// TwinCAT 3 PLC project MS
// ProgramVersion: 3.1.4024.0
// libraries:
//   Tc2_ControllerToolbox, * (Beckhoff Automation GmbH)
//   Tc2_ModbusRTU, * (Beckhoff Automation GmbH)
//   Tc2_SerialCom, * (Beckhoff Automation GmbH)
//   Tc2_Standard, * (Beckhoff Automation GmbH)
//   Tc2_System, * (Beckhoff Automation GmbH)
//   Tc2_Utilities, * (Beckhoff Automation GmbH)
//   Tc3_Module, * (Beckhoff Automation GmbH)
// project tree:
//   DATA TYPES/MODUELS/ ST_GAS_CABINET.TcDUT (not stored), ST_MAIN_MODULE.TcDUT (not stored), ST_NOTIFICATION.TcDUT (not stored), ST_NOTIFICATION_MESSAGE.TcDUT (not stored), ST_REACTOR_CABINET.TcDUT (not stored), ST_SEQUENCE.TcDUT (not stored), ST_SOL_VALVE.TcDUT (not stored), ST_TEMP_CONTROLLER.TcDUT (not stored), ST_THROTTLE_VALVE.TcDUT (not stored)
//   DATA TYPES/PARTS/ ST_ANALOG_PART.TcDUT (not stored), ST_DIGITAL_PART.TcDUT (not stored), ST_SEQUENCE_PART.TcDUT (not stored)
//   DEVICE/LINE HEATER/ FB_LINE_HEATER_MANAGER.TcPOU (not stored), FB_Modbus_Send_FIFO.TcPOU (not stored), FB_TEMP_RAMPING.TcPOU (not stored)
//   DEVICE/LINE HEATER/FUNCTION/ F_Temp_Write_Set_Point.TcPOU (not stored), F_Temp_Write_Value.TcPOU (not stored)
//   DEVICE/ ST_LineHeater_Data.TcDUT (not stored), ST_Modbus_Send_Frame.TcDUT (not stored)
//   DUTs/DUTs/ENUM/ E_aAnalogInputIO_Index.TcDUT, E_AlarmList.TcDUT (not stored), E_AlarmSetValue.TcDUT, E_InputState.TcDUT (not stored), E_Interlock.TcDUT (not stored), E_Morning_Index.TcDUT, E_WarningList.TcDUT (not stored)
//   DUTs/DUTs/ F_GetReal_USINT.TcDUT (not stored)
//   DUTs/ E_ControlMode.TcDUT (not stored), E_RampGeneratorState.TcDUT (not stored), E_RecipeRun.TcDUT (not stored), E_RecipeRunETMode.TcDUT (not stored), E_TowerLamp.TcDUT (not stored), OperationMode.TcDUT (not stored), outWord.TcDUT (not stored), RampGeneratorInput.TcDUT (not stored), RecipeRunET.TcDUT (not stored), RecipeStep.TcDUT, ScaleFactor.TcDUT (not stored)
//   FUNCTION/ BOOL_TO_STRING_LHeaterON.TcPOU (not stored), CheckRangeSigned.TcPOU (not stored), CheckRangeUnsigned.TcPOU (not stored), FB_TON_Pausable.TcPOU (not stored), F_GetDorPressure.TcPOU, F_State_All_Valve_Vent.TcPOU (not stored), HEXSTR_TO_REAL_LHeaterPV.TcPOU (not stored), Real_To_String_LineHeater.TcPOU (not stored), Real_To_String_ThermalBath.TcPOU (not stored), USINT_TO_WORD_Bit.TcPOU (not stored), USINT_TO_WORD_jh.TcPOU (not stored), WORD_TO_USINT_Bit.TcPOU (not stored)
//   GVLs/ GVL_COMMAND_FROM_UI.TcGVL (not stored), GVL_CONSTANT.TcGVL, GVL_DEVICE_NET_E3508.TcGVL, GVL_DEVICE_NET_IQ_PLUS.TcGVL (not stored), GVL_IO.TcGVL, GVL.TcGVL, GVL_IO_GAS_CABINET.TcGVL (not stored), GVL_IO_REACTOR_CABINET.TcGVL (not stored), GVL_IO_VALVE.TcGVL (not stored), GVL_PERSISTENT.TcGVL (not stored), GVL_SEQUENCE.TcGVL, GVL_Serial.TcGVL, RCP.TcGVL (not stored)
//   / PlcTask.TcTTO (not stored)
//   POUs/ FB_AnalogDeviceRampControl.TcPOU, FB_ControlRampGenerator.TcPOU (not stored), FB_DeviationCheck.TcPOU, FB_FaultCheck.TcPOU (not stored), FB_OnlyPVUpdate.TcPOU, FB_OverLimitCheck.TcPOU (not stored), FB_RecipeAnalogControlInputSequencer.TcPOU, F_StopAnalogRamping_ForRecipe.TcPOU, FB_SensorLimitCheck.TcPOU (not stored), FB_ValveControl.TcPOU, F_ResetTimersAndRCPTimes.TcPOU (not stored), MAIN.TcPOU, P11_E3508.TcPOU, P12_IQ_PLUS.TcPOU, P13_LineHeater.TcPOU, P14_ThermalBath.TcPOU, P15_RotationOperation.TcPOU, P16_CoverOperation.TcPOU, P17_DOROperation.TcPOU, P22_Background_ThermalBath.TcPOU (not stored), P30_ManualControl.TcPOU, P31_PriorityControl.TcPOU (not stored), P50_RecipeControl.TcPOU, P70_Interface.TcPOU, P90_Interlock.TcPOU, P91_Monitoring.TcPOU, P92_Maintenance.TcPOU
//   POUs/FUNCTION/ FB_RINGBUFFER.TcPOU (not stored), F_StateValve_Process_Source.TcPOU (not stored), F_StateValve_Process.TcPOU (not stored)
//   POUs/VARIABLE_LINK/ F_Variable_DeviceLink.TcPOU, F_Variable_Valve.TcPOU, F_Variable_FromUI.TcPOU, F_Variable_FromUI_Interlock.TcPOU, F_Variable_TODevice.TcPOU (not stored), F_Variable_ToUI_InputState.TcPOU
// real-time tasks:
//   TASK PlcTask: cycle T#10ms, priority 20, ADS port 350
// I/O:
//   DEVICE Device 1 (EtherCAT), AmsNetId 10.10.10.10.2.1
//     Term 1 (EK1200) [EK1200-5000 EtherCAT Power supply (2A E-Bus)]
//       Term 2 (EL1088) [EL1088 8Ch. Dig. Input 24V, 3ms, negative]
//       Term 3 (EL1088) [EL1088 8Ch. Dig. Input 24V, 3ms, negative]
//       Term 4 (EL1088) [EL1088 8Ch. Dig. Input 24V, 3ms, negative]
//       Term 5 (EL1088) [EL1088 8Ch. Dig. Input 24V, 3ms, negative]
//       Term 6 (EL1088) [EL1088 8Ch. Dig. Input 24V, 3ms, negative]
//       Term 7 (EL1088) [EL1088 8Ch. Dig. Input 24V, 3ms, negative]
//       Term 8 (EL2088) [EL2088 8Ch. Dig. Output 24V, 0.5A, switching to negative]
//       Term 9 (EL2088) [EL2088 8Ch. Dig. Output 24V, 0.5A, switching to negative]
//       Term 10 (EL3064) [EL3064 4Ch. Ana. Input 0-10V]
//       Term 11 (EL4004) [EL4004 4Ch. Ana. Output 0-10V, 12bit]
//       Term 12 (EL9410) [EL9410 E-Bus Power Supplier  (Diagnostics)]
//       Term 13 (EL3064) [EL3064 4Ch. Ana. Input 0-10V]
//       Term 14 (EL4004) [EL4004 4Ch. Ana. Output 0-10V, 12bit]
//       Term 15 (EL3064) [EL3064 4Ch. Ana. Input 0-10V]
//       Term 16 (EL4004) [EL4004 4Ch. Ana. Output 0-10V, 12bit]
//       Term 17 (EL3064) [EL3064 4Ch. Ana. Input 0-10V]
//       Term 18 (EL4004) [EL4004 4Ch. Ana. Output 0-10V, 12bit]
//       Term 19 (EL3102) [EL3102 2Ch. Ana. Input +/-10V, Diff.]
//       Term 20 (EL3024) [EL3024 4Ch. Ana. Input 4-20mA DIFF]
//       Term 21 (EL6021) [EL6021 Interface (RS422/485)]
//       Term 22 (EL6021) [EL6021 Interface (RS422/485)]
//       Term 23 (EL6752) [EL6752 DeviceNet Master]
//       Term 24 (EK1110) [EK1110 EtherCAT extension]
//     Term 25 (EK1100) [EK1100 EtherCAT Coupler (2A E-Bus)]
//       Term 26 (EL1088) [EL1088 8Ch. Dig. Input 24V, 3ms, negative]
//       Term 27 (EL1088) [EL1088 8Ch. Dig. Input 24V, 3ms, negative]
//       Term 28 (EL1088) [EL1088 8Ch. Dig. Input 24V, 3ms, negative]
//       Term 29 (EL2088) [EL2088 8Ch. Dig. Output 24V, 0.5A, switching to negative]
//       Term 30 (EL2088) [EL2088 8Ch. Dig. Output 24V, 0.5A, switching to negative]
//       Term 31 (EL2088) [EL2088 8Ch. Dig. Output 24V, 0.5A, switching to negative]
//       Term 32 (EL3064) [EL3064 4Ch. Ana. Input 0-10V]
//       Term 33 (EL3024) [EL3024 4Ch. Ana. Input 4-20mA DIFF]
//       Term 34 (EL4004) [EL4004 4Ch. Ana. Output 0-10V, 12bit]
//       Term 35 (EL3204) [EL3204 4Ch. Ana. Input PT100 (RTD)]
//       Term 36 (EL9011) [EL9011 End Terminal]
//   DEVICE Device 2 (EL6752), AmsNetId 10.10.10.10.3.1
//     SolValve // EDS-File: 'OPP6-2D.EDS' DescText: OPP6-2D Vendor: CKD Corporation Device Type: Generic Device Product Name: OPP6-2D Catalog Number:
//     ThrottleValve // EDS-File: 'TBJQPDNG-L041X01 155OUT154.EDS' DescText: Intellisys IQ-Plus Vendor: Nor-Cal Products Device Type: Process Control Valve Product Name: INTELLISYS Catalog Number: IQ-Plus
//     TempController // EDS-File: '3500-2.3V2.EDS' DescText: Eurotherm 3500 Vendor: Eurotherm Device Type: Generic Product Name: Eurotherm 3500 Catalog Number:
// variable links:
//   MS/MS Instance <-> Device 1 (EtherCAT)/Term 1 (EK1200)/Term 10 (EL3064)
//     PlcTask Inputs/GVL_IO_GAS_CABINET.AI_09_M01_ChalcogenRunPV <-> AI Standard Channel 1/Value
//     PlcTask Inputs/GVL_IO_GAS_CABINET.AI_09_M02_MORunPV <-> AI Standard Channel 2/Value
//     PlcTask Inputs/GVL_IO_GAS_CABINET.AI_09_M03_H2SeSupplyPV <-> AI Standard Channel 3/Value
//     PlcTask Inputs/GVL_IO_GAS_CABINET.AI_09_M04_H2SSupplyPV <-> AI Standard Channel 4/Value
//   MS/MS Instance <-> Device 1 (EtherCAT)/Term 1 (EK1200)/Term 11 (EL4004)
//     PlcTask Outputs/GVL_IO_GAS_CABINET.AO_10_M01_ChalcogenRunSV <-> AO Outputs Channel 1/Analog output
//     PlcTask Outputs/GVL_IO_GAS_CABINET.AO_10_M02_MORunSV <-> AO Outputs Channel 2/Analog output
//     PlcTask Outputs/GVL_IO_GAS_CABINET.AO_10_M03_H2SeSupplySV <-> AO Outputs Channel 3/Analog output
//     PlcTask Outputs/GVL_IO_GAS_CABINET.AO_10_M04_H2SSupplySV <-> AO Outputs Channel 4/Analog output
//   MS/MS Instance <-> Device 1 (EtherCAT)/Term 1 (EK1200)/Term 13 (EL3064)
//     PlcTask Inputs/GVL_IO_GAS_CABINET.AI_11_M05_Source_1TMInSupplyPV <-> AI Standard Channel 1/Value
//     PlcTask Inputs/GVL_IO_GAS_CABINET.AI_11_M06_Source_2TMGaSupplyPV <-> AI Standard Channel 2/Value
//     PlcTask Inputs/GVL_IO_GAS_CABINET.AI_11_M07_Source_3DMSeSupplyPV <-> AI Standard Channel 3/Value
//     PlcTask Inputs/GVL_IO_GAS_CABINET.AI_11_M08_Source_4ChalcoSupplyPV <-> AI Standard Channel 4/Value
//   MS/MS Instance <-> Device 1 (EtherCAT)/Term 1 (EK1200)/Term 14 (EL4004)
//     PlcTask Outputs/GVL_IO_GAS_CABINET.AO_12_M05_Source_1TMInSupplySV <-> AO Outputs Channel 1/Analog output
//     PlcTask Outputs/GVL_IO_GAS_CABINET.AO_12_M06_Source_2TMGaSupplySV <-> AO Outputs Channel 2/Analog output
//     PlcTask Outputs/GVL_IO_GAS_CABINET.AO_12_M07_Source_3DMSeSupplySV <-> AO Outputs Channel 3/Analog output
//     PlcTask Outputs/GVL_IO_GAS_CABINET.AO_12_M08_Source_4ChalcoSupplySV <-> AO Outputs Channel 4/Analog output
//   MS/MS Instance <-> Device 1 (EtherCAT)/Term 1 (EK1200)/Term 15 (EL3064)
//     PlcTask Inputs/GVL_IO_GAS_CABINET.AI_13_M09_LinerPurgePV <-> AI Standard Channel 1/Value
//     PlcTask Inputs/GVL_IO_GAS_CABINET.AI_13_M10_HeaterPurgePV <-> AI Standard Channel 2/Value
//     PlcTask Inputs/GVL_IO_GAS_CABINET.AI_13_M11_ChalcogenVentPV <-> AI Standard Channel 3/Value
//     PlcTask Inputs/GVL_IO_GAS_CABINET.AI_13_M12_MOVentPV <-> AI Standard Channel 4/Value
//   MS/MS Instance <-> Device 1 (EtherCAT)/Term 1 (EK1200)/Term 16 (EL4004)
//     PlcTask Outputs/GVL_IO_GAS_CABINET.AO_14_M09_LinerPurgeSV <-> AO Outputs Channel 1/Analog output
//     PlcTask Outputs/GVL_IO_GAS_CABINET.AO_14_M10_HeaterPurgeSV <-> AO Outputs Channel 2/Analog output
//     PlcTask Outputs/GVL_IO_GAS_CABINET.AO_14_M11_ChalcogenVentSV <-> AO Outputs Channel 3/Analog output
//     PlcTask Outputs/GVL_IO_GAS_CABINET.AO_14_M12_MOVentSV <-> AO Outputs Channel 4/Analog output
//   MS/MS Instance <-> Device 1 (EtherCAT)/Term 1 (EK1200)/Term 17 (EL3064)
//     PlcTask Inputs/GVL_IO_GAS_CABINET.AI_15_E01Source_1TMInPressurePV <-> AI Standard Channel 1/Value
//     PlcTask Inputs/GVL_IO_GAS_CABINET.AI_15_E02Source_2TMGaPressurePV <-> AI Standard Channel 2/Value
//     PlcTask Inputs/GVL_IO_GAS_CABINET.AI_15_E03Source_3DMSePressurePV <-> AI Standard Channel 3/Value
//     PlcTask Inputs/GVL_IO_GAS_CABINET.AI_15_E04Source_4ChalcoPressurePV <-> AI Standard Channel 4/Value
//   MS/MS Instance <-> Device 1 (EtherCAT)/Term 1 (EK1200)/Term 18 (EL4004)
//     PlcTask Outputs/GVL_IO_GAS_CABINET.AO_16_E01Source_1TMInPressureSV <-> AO Outputs Channel 1/Analog output
//     PlcTask Outputs/GVL_IO_GAS_CABINET.AO_16_E02Source_2TMGaPressureSV <-> AO Outputs Channel 2/Analog output
//     PlcTask Outputs/GVL_IO_GAS_CABINET.AO_16_E03Source_3DMSePressureSV <-> AO Outputs Channel 3/Analog output
//     PlcTask Outputs/GVL_IO_GAS_CABINET.AO_16_E04Source_4ChalcoPressureSV <-> AO Outputs Channel 4/Analog output
//   MS/MS Instance <-> Device 1 (EtherCAT)/Term 1 (EK1200)/Term 19 (EL3102)
//     PlcTask Inputs/GVL_IO_GAS_CABINET.DI_17_DP1ChalcogenDP <-> AI Standard Channel 1/Value
//     PlcTask Inputs/GVL_IO_GAS_CABINET.DI_17_DP2MODP <-> AI Standard Channel 2/Value
//   MS/MS Instance <-> Device 1 (EtherCAT)/Term 1 (EK1200)/Term 2 (EL1088)
//     PlcTask Inputs/GVL_IO_GAS_CABINET.DI_01_ControlCabinetDoorClose <-> Channel 5/Input
//     PlcTask Inputs/GVL_IO_GAS_CABINET.DI_01_GasCabinetDoorClose <-> Channel 4/Input
//     PlcTask Inputs/GVL_IO_GAS_CABINET.DI_01_GasCabinetLampButton <-> Channel 2/Input
//     PlcTask Inputs/GVL_IO_GAS_CABINET.DI_01_PneumaticPressureSensor <-> Channel 3/Input
//     PlcTask Inputs/GVL_IO_GAS_CABINET.DI_01_ResetButton <-> Channel 1/Input
//     PlcTask Inputs/GVL_IO_GAS_CABINET.DI_01_SMPS_1Alarm <-> Channel 6/Input
//     PlcTask Inputs/GVL_IO_GAS_CABINET.DI_01_SMPS_2Alarm <-> Channel 7/Input
//     PlcTask Inputs/GVL_IO_GAS_CABINET.DI_01_SMPS_3Alarm <-> Channel 8/Input
//   MS/MS Instance <-> Device 1 (EtherCAT)/Term 1 (EK1200)/Term 20 (EL3024)
//     PlcTask Inputs/GVL_IO_GAS_CABINET.DI_18_S01N2SupplyPressPV <-> AI Standard Channel 1/Value
//     PlcTask Inputs/GVL_IO_GAS_CABINET.DI_18_S02H2SupplyPressPV <-> AI Standard Channel 2/Value
//     PlcTask Inputs/GVL_IO_GAS_CABINET.DI_18_S03H2SSupplyPressPV <-> AI Standard Channel 3/Value
//     PlcTask Inputs/GVL_IO_GAS_CABINET.DI_18_S04H2SeSupplyPressPV <-> AI Standard Channel 4/Value
//   MS/MS Instance <-> Device 1 (EtherCAT)/Term 1 (EK1200)/Term 21 (EL6021)
//     PlcTask Inputs/GVL.fbLineHeater_Manager.fbModbus_Master.InData/D <-> COM TxPDO-Map Inputs/Data In 0
//     PlcTask Inputs/GVL.fbLineHeater_Manager.fbModbus_Master.InData/D @bit {8..168 step 8} <-> COM TxPDO-Map Inputs/Data In {1..21}  (21 links)
//     PlcTask Inputs/GVL.fbLineHeater_Manager.fbModbus_Master.InData/Status <-> COM TxPDO-Map Inputs/Status
//     PlcTask Outputs/GVL.fbLineHeater_Manager.fbModbus_Master.OutData/Ctrl <-> COM RxPDO-Map Outputs/Ctrl
//     PlcTask Outputs/GVL.fbLineHeater_Manager.fbModbus_Master.OutData/D <-> COM RxPDO-Map Outputs/Data Out 0
//     PlcTask Outputs/GVL.fbLineHeater_Manager.fbModbus_Master.OutData/D @bit {8..168 step 8} <-> COM RxPDO-Map Outputs/Data Out {1..21}  (21 links)
//   MS/MS Instance <-> Device 1 (EtherCAT)/Term 1 (EK1200)/Term 22 (EL6021)
//     PlcTask Inputs/GVL_Serial.stIn_KL6031_TB/D <-> COM TxPDO-Map Inputs/Data In 0
//     PlcTask Inputs/GVL_Serial.stIn_KL6031_TB/D @bit {8..168 step 8} <-> COM TxPDO-Map Inputs/Data In {1..21}  (21 links)
//     PlcTask Inputs/GVL_Serial.stIn_KL6031_TB/Status <-> COM TxPDO-Map Inputs/Status
//     PlcTask Outputs/GVL_Serial.stOut_KL6031_TB/Ctrl <-> COM RxPDO-Map Outputs/Ctrl
//     PlcTask Outputs/GVL_Serial.stOut_KL6031_TB/D <-> COM RxPDO-Map Outputs/Data Out 0
//     PlcTask Outputs/GVL_Serial.stOut_KL6031_TB/D @bit {8..168 step 8} <-> COM RxPDO-Map Outputs/Data Out {1..21}  (21 links)
//   MS/MS Instance <-> Device 1 (EtherCAT)/Term 1 (EK1200)/Term 3 (EL1088)
//     PlcTask Inputs/GVL_IO_GAS_CABINET.DI_02_CoverLiftMotorCP <-> Channel 7/Input
//     PlcTask Inputs/GVL_IO_GAS_CABINET.DI_02_GraphiteHeaterELCB <-> Channel 2/Input
//     PlcTask Inputs/GVL_IO_GAS_CABINET.DI_02_LineHeatersELCB <-> Channel 5/Input
//     PlcTask Inputs/GVL_IO_GAS_CABINET.DI_02_RotationMotorCP <-> Channel 6/Input
//     PlcTask Inputs/GVL_IO_GAS_CABINET.DI_02_SMPS_4Alarm <-> Channel 1/Input
//     PlcTask Inputs/GVL_IO_GAS_CABINET.DI_02_T_VCP <-> Channel 8/Input
//     PlcTask Inputs/GVL_IO_GAS_CABINET.DI_02_ThermalBathsELCB <-> Channel 3/Input
//     PlcTask Inputs/GVL_IO_GAS_CABINET.DI_02_VacuumPumpELCB <-> Channel 4/Input
//   MS/MS Instance <-> Device 1 (EtherCAT)/Term 1 (EK1200)/Term 4 (EL1088)
//     PlcTask Inputs/GVL_IO_GAS_CABINET.DI_03_CabinetLampsCP <-> Channel 2/Input
//     PlcTask Inputs/GVL_IO_GAS_CABINET.DI_03_GasDetectorCP <-> Channel 1/Input
//     PlcTask Inputs/GVL_IO_GAS_CABINET.DI_03_LineHeater_1CP <-> Channel 4/Input
//     PlcTask Inputs/GVL_IO_GAS_CABINET.DI_03_LineHeater_2CP <-> Channel 5/Input
//     PlcTask Inputs/GVL_IO_GAS_CABINET.DI_03_LineHeater_3CP <-> Channel 6/Input
//     PlcTask Inputs/GVL_IO_GAS_CABINET.DI_03_LineHeater_4CP <-> Channel 7/Input
//     PlcTask Inputs/GVL_IO_GAS_CABINET.DI_03_LineHeater_5CP <-> Channel 8/Input
//     PlcTask Inputs/GVL_IO_GAS_CABINET.DI_03_MFCPowerCP <-> Channel 3/Input
//   MS/MS Instance <-> Device 1 (EtherCAT)/Term 1 (EK1200)/Term 5 (EL1088)
//     PlcTask Inputs/GVL_IO_GAS_CABINET.DI_04_ExternalScrubberFault <-> Channel 8/Input
//     PlcTask Inputs/GVL_IO_GAS_CABINET.DI_04_FireSensor <-> Channel 7/Input
//     PlcTask Inputs/GVL_IO_GAS_CABINET.DI_04_GasDetectorH2 <-> Channel 4/Input
//     PlcTask Inputs/GVL_IO_GAS_CABINET.DI_04_GasDetectorH2S <-> Channel 5/Input
//     PlcTask Inputs/GVL_IO_GAS_CABINET.DI_04_GasDetectorH2Se <-> Channel 6/Input
//     PlcTask Inputs/GVL_IO_GAS_CABINET.DI_04_LineHeater_6CP <-> Channel 1/Input
//     PlcTask Inputs/GVL_IO_GAS_CABINET.DI_04_LineHeater_7CP <-> Channel 2/Input
//     PlcTask Inputs/GVL_IO_GAS_CABINET.DI_04_LineHeater_8CP <-> Channel 3/Input
//   MS/MS Instance <-> Device 1 (EtherCAT)/Term 1 (EK1200)/Term 6 (EL1088)
//     PlcTask Inputs/GVL_IO_GAS_CABINET.DI_05_ExternalH2GasCabinetFault <-> Channel 1/Input
//     PlcTask Inputs/GVL_IO_GAS_CABINET.DI_05_ExternalH2SGasCabinetFault <-> Channel 2/Input
//     PlcTask Inputs/GVL_IO_GAS_CABINET.DI_05_ExternalH2SeGasCabinetFault <-> Channel 3/Input
//     PlcTask Inputs/GVL_IO_GAS_CABINET.DI_05_ExternalUserInputAlarm <-> Channel 4/Input
//     PlcTask Inputs/GVL_IO_GAS_CABINET.DI_05_ThermalBath_1CutOffAlarm <-> Channel 6/Input
//     PlcTask Inputs/GVL_IO_GAS_CABINET.DI_05_ThermalBath_2CutOffAlarm <-> Channel 8/Input
//     PlcTask Inputs/GVL_IO_GAS_CABINET.DI_05_ThermalBath_1DeviationAlarm <-> Channel 5/Input
//     PlcTask Inputs/GVL_IO_GAS_CABINET.DI_05_ThermalBath_2DeviationAlarm <-> Channel 7/Input
//   MS/MS Instance <-> Device 1 (EtherCAT)/Term 1 (EK1200)/Term 7 (EL1088)
//     PlcTask Inputs/GVL_IO_GAS_CABINET.DI_06_Spare_01 <-> Channel 5/Input
//     PlcTask Inputs/GVL_IO_GAS_CABINET.DI_06_Spare_02 <-> Channel 6/Input
//     PlcTask Inputs/GVL_IO_GAS_CABINET.DI_06_Spare_03 <-> Channel 7/Input
//     PlcTask Inputs/GVL_IO_GAS_CABINET.DI_06_Spare_04 <-> Channel 8/Input
//     PlcTask Inputs/GVL_IO_GAS_CABINET.DI_06_ThermalBath_3CutOffAlarm <-> Channel 2/Input
//     PlcTask Inputs/GVL_IO_GAS_CABINET.DI_06_ThermalBath_4CutOffAlarm <-> Channel 4/Input
//     PlcTask Inputs/GVL_IO_GAS_CABINET.DI_06_ThermalBath_3DeviationAlarm <-> Channel 1/Input
//     PlcTask Inputs/GVL_IO_GAS_CABINET.DI_06_ThermalBath_4DeviationAlarm <-> Channel 3/Input
//   MS/MS Instance <-> Device 1 (EtherCAT)/Term 1 (EK1200)/Term 8 (EL2088)
//     PlcTask Outputs/GVL_IO_GAS_CABINET.DO_07_ControlCabinetLamp <-> Channel 2/Output
//     PlcTask Outputs/GVL_IO_GAS_CABINET.DO_07_GasCabinetLamp <-> Channel 3/Output
//     PlcTask Outputs/GVL_IO_GAS_CABINET.DO_07_GraphiteHeaterMC <-> Channel 4/Output
//     PlcTask Outputs/GVL_IO_GAS_CABINET.DO_07_LineHeatersMC <-> Channel 7/Output
//     PlcTask Outputs/GVL_IO_GAS_CABINET.DO_07_ResetButtonLamp <-> Channel 8/Output
//     PlcTask Outputs/GVL_IO_GAS_CABINET.DO_07_SystemPowerOffLock <-> Channel 1/Output
//     PlcTask Outputs/GVL_IO_GAS_CABINET.DO_07_ThermalBathsMC <-> Channel 5/Output
//     PlcTask Outputs/GVL_IO_GAS_CABINET.DO_07_VacuumPumpMC <-> Channel 6/Output
//   MS/MS Instance <-> Device 1 (EtherCAT)/Term 1 (EK1200)/Term 9 (EL2088)
//     PlcTask Outputs/GVL_IO_GAS_CABINET.DO_08_Spare_01 <-> Channel 1/Output
//     PlcTask Outputs/GVL_IO_GAS_CABINET.DO_08_Spare_02 <-> Channel 2/Output
//     PlcTask Outputs/GVL_IO_GAS_CABINET.DO_08_Spare_03 <-> Channel 3/Output
//     PlcTask Outputs/GVL_IO_GAS_CABINET.DO_08_Spare_04 <-> Channel 4/Output
//     PlcTask Outputs/GVL_IO_GAS_CABINET.DO_08_Spare_05 <-> Channel 5/Output
//     PlcTask Outputs/GVL_IO_GAS_CABINET.DO_08_Spare_06 <-> Channel 6/Output
//     PlcTask Outputs/GVL_IO_GAS_CABINET.DO_08_Spare_07 <-> Channel 7/Output
//     PlcTask Outputs/GVL_IO_GAS_CABINET.DO_08_Spare_08 <-> Channel 8/Output
//   MS/MS Instance <-> Device 1 (EtherCAT)/Term 25 (EK1100)/Term 26 (EL1088)
//     PlcTask Inputs/GVL_IO_REACTOR_CABINET.DI_01_ClampLock <-> Channel 7/Input
//     PlcTask Inputs/GVL_IO_REACTOR_CABINET.DI_01_ClampRelease <-> Channel 8/Input
//     PlcTask Inputs/GVL_IO_REACTOR_CABINET.DI_01_DORATMButton <-> Channel 4/Input
//     PlcTask Inputs/GVL_IO_REACTOR_CABINET.DI_01_DORVACButton <-> Channel 3/Input
//     PlcTask Inputs/GVL_IO_REACTOR_CABINET.DI_01_MaintenanceModeKey <-> Channel 1/Input
//     PlcTask Inputs/GVL_IO_REACTOR_CABINET.DI_01_ReactorCabinetLampButton <-> Channel 2/Input
//     PlcTask Inputs/GVL_IO_REACTOR_CABINET.DI_01_ReactorDoorDownButton <-> Channel 6/Input
//     PlcTask Inputs/GVL_IO_REACTOR_CABINET.DI_01_ReactorDoorUpButton <-> Channel 5/Input
//   MS/MS Instance <-> Device 1 (EtherCAT)/Term 25 (EK1100)/Term 27 (EL1088)
//     PlcTask Inputs/GVL_IO_REACTOR_CABINET.DI_02_C_WFlowSensor <-> Channel 1/Input
//     PlcTask Inputs/GVL_IO_REACTOR_CABINET.DI_02_ReactorDoorUpLimitSensor <-> Channel 8/Input
//     PlcTask Inputs/GVL_IO_REACTOR_CABINET.DI_02_SusceptorRotationMotorFault <-> Channel 2/Input
//     PlcTask Inputs/GVL_IO_REACTOR_CABINET.DI_02_VacuumPumpAlarm <-> Channel 5/Input
//     PlcTask Inputs/GVL_IO_REACTOR_CABINET.DI_02_VacuumPumpFBRunning <-> Channel 7/Input
//     PlcTask Inputs/GVL_IO_REACTOR_CABINET.DI_02_VacuumPumpFail <-> Channel 3/Input
//     PlcTask Inputs/GVL_IO_REACTOR_CABINET.DI_02_VacuumPumpRunning <-> Channel 6/Input
//     PlcTask Inputs/GVL_IO_REACTOR_CABINET.DI_02_VacuumPumpWarning <-> Channel 4/Input
//   MS/MS Instance <-> Device 1 (EtherCAT)/Term 25 (EK1100)/Term 28 (EL1088)
//     PlcTask Inputs/GVL_IO_REACTOR_CABINET.DI_03_CylinderAutoSwitch_Closed <-> Channel 2/Input
//     PlcTask Inputs/GVL_IO_REACTOR_CABINET.DI_03_CylinderAutoSwitch_Opened <-> Channel 3/Input
//     PlcTask Inputs/GVL_IO_REACTOR_CABINET.DI_03_ReactorCabinetDoorClose <-> Channel 4/Input
//     PlcTask Inputs/GVL_IO_REACTOR_CABINET.DI_03_ReactorDoorDownLimitSensor <-> Channel 1/Input
//     PlcTask Inputs/GVL_IO_REACTOR_CABINET.DI_03_Spare_01 <-> Channel 5/Input
//     PlcTask Inputs/GVL_IO_REACTOR_CABINET.DI_03_Spare_02 <-> Channel 6/Input
//     PlcTask Inputs/GVL_IO_REACTOR_CABINET.DI_03_Spare_03 <-> Channel 7/Input
//     PlcTask Inputs/GVL_IO_REACTOR_CABINET.DI_03_Spare_04 <-> Channel 8/Input
//   MS/MS Instance <-> Device 1 (EtherCAT)/Term 25 (EK1100)/Term 29 (EL2088)
//     PlcTask Outputs/GVL_IO_REACTOR_CABINET.DO_04_ReactorCoverDownRelay <-> Channel 8/Output
//     PlcTask Outputs/GVL_IO_REACTOR_CABINET.DO_04_ReactorCoverUpRelay <-> Channel 7/Output
//     PlcTask Outputs/GVL_IO_REACTOR_CABINET.DO_04_SignalTowerBlue <-> Channel 4/Output
//     PlcTask Outputs/GVL_IO_REACTOR_CABINET.DO_04_SignalTowerBuzzer <-> Channel 6/Output
//     PlcTask Outputs/GVL_IO_REACTOR_CABINET.DO_04_SignalTowerGreen <-> Channel 3/Output
//     PlcTask Outputs/GVL_IO_REACTOR_CABINET.DO_04_SignalTowerOrange <-> Channel 2/Output
//     PlcTask Outputs/GVL_IO_REACTOR_CABINET.DO_04_SignalTowerRed <-> Channel 1/Output
//     PlcTask Outputs/GVL_IO_REACTOR_CABINET.DO_04_SignalTowerWhite <-> Channel 5/Output
//   MS/MS Instance <-> Device 1 (EtherCAT)/Term 25 (EK1100)/Term 30 (EL2088)
//     PlcTask Outputs/GVL_IO_REACTOR_CABINET.DO_05_ClampLock <-> Channel 1/Output
//     PlcTask Outputs/GVL_IO_REACTOR_CABINET.DO_05_ClampRelease <-> Channel 2/Output
//     PlcTask Outputs/GVL_IO_REACTOR_CABINET.DO_05_DORVACButtonLamp <-> Channel 8/Output
//     PlcTask Outputs/GVL_IO_REACTOR_CABINET.DO_05_SusceptorRotationAL_RST <-> Channel 7/Output
//     PlcTask Outputs/GVL_IO_REACTOR_CABINET.DO_05_SusceptorRotationFWD <-> Channel 5/Output
//     PlcTask Outputs/GVL_IO_REACTOR_CABINET.DO_05_SusceptorRotationSTOP <-> Channel 6/Output
//     PlcTask Outputs/GVL_IO_REACTOR_CABINET.DO_05_VacuumPumpReset <-> Channel 4/Output
//     PlcTask Outputs/GVL_IO_REACTOR_CABINET.DO_05_VacuumPumpStart_Stop <-> Channel 3/Output
//   MS/MS Instance <-> Device 1 (EtherCAT)/Term 25 (EK1100)/Term 31 (EL2088)
//     PlcTask Outputs/GVL_IO_REACTOR_CABINET.DO_06_ClampLockButtonLamp <-> Channel 4/Output
//     PlcTask Outputs/GVL_IO_REACTOR_CABINET.DO_06_ClampReleaseButtonLamp <-> Channel 5/Output
//     PlcTask Outputs/GVL_IO_REACTOR_CABINET.DO_06_DORATMButtonLamp <-> Channel 1/Output
//     PlcTask Outputs/GVL_IO_REACTOR_CABINET.DO_06_ReactorCabinetLamp <-> Channel 6/Output
//     PlcTask Outputs/GVL_IO_REACTOR_CABINET.DO_06_ReactorCoverDownButtonLamp <-> Channel 3/Output
//     PlcTask Outputs/GVL_IO_REACTOR_CABINET.DO_06_ReactorCoverUpButtonLamp <-> Channel 2/Output
//     PlcTask Outputs/GVL_IO_REACTOR_CABINET.DO_06_Spare07 <-> Channel 7/Output
//     PlcTask Outputs/GVL_IO_REACTOR_CABINET.DO_06_Spare08 <-> Channel 8/Output
//   MS/MS Instance <-> Device 1 (EtherCAT)/Term 25 (EK1100)/Term 32 (EL3064)
//     PlcTask Inputs/GVL_IO_REACTOR_CABINET.AI_07_P02_ReactorPressure10TorrPV <-> AI Standard Channel 1/Value
//     PlcTask Inputs/GVL_IO_REACTOR_CABINET.AI_07_P03_ExhaustPressurePV <-> AI Standard Channel 3/Value
//     PlcTask Inputs/GVL_IO_REACTOR_CABINET.AI_07_S05_DORPressurePV <-> AI Standard Channel 2/Value
//     PlcTask Inputs/GVL_IO_REACTOR_CABINET.AI_07_Spare_04 <-> AI Standard Channel 4/Value
//   MS/MS Instance <-> Device 1 (EtherCAT)/Term 25 (EK1100)/Term 33 (EL3024)
//     PlcTask Inputs/GVL_IO_REACTOR_CABINET.AI_08_R01SusceptorRotationPV <-> AI Standard Channel 1/Value
//     PlcTask Inputs/GVL_IO_REACTOR_CABINET.AI_08_Spare_02 <-> AI Standard Channel 2/Value
//     PlcTask Inputs/GVL_IO_REACTOR_CABINET.AI_08_Spare_03 <-> AI Standard Channel 3/Value
//     PlcTask Inputs/GVL_IO_REACTOR_CABINET.AI_08_Spare_04 <-> AI Standard Channel 4/Value
//   MS/MS Instance <-> Device 1 (EtherCAT)/Term 25 (EK1100)/Term 34 (EL4004)
//     PlcTask Outputs/GVL_IO_REACTOR_CABINET.AO_09_P03_ExhaustPressureAM215Input <-> AO Outputs Channel 1/Analog output
//     PlcTask Outputs/GVL_IO_REACTOR_CABINET.AO_09_R01_SusceptorRotationSV <-> AO Outputs Channel 2/Analog output
//     PlcTask Outputs/GVL_IO_REACTOR_CABINET.AO_09_Spare_03 <-> AO Outputs Channel 3/Analog output
//     PlcTask Outputs/GVL_IO_REACTOR_CABINET.AO_09_Spare_04 <-> AO Outputs Channel 4/Analog output
//   MS/MS Instance <-> Device 1 (EtherCAT)/Term 25 (EK1100)/Term 35 (EL3204)
//     PlcTask Inputs/GVL_IO_REACTOR_CABINET.AI_10_R04S_HCoolingWaterPV <-> RTD Inputs Channel 1/Value
//     PlcTask Inputs/GVL_IO_REACTOR_CABINET.AI_10_Spare_02 <-> RTD Inputs Channel 2/Value
//     PlcTask Inputs/GVL_IO_REACTOR_CABINET.AI_10_Spare_03 <-> RTD Inputs Channel 3/Value
//     PlcTask Inputs/GVL_IO_REACTOR_CABINET.AI_10_Spare_04 <-> RTD Inputs Channel 4/Value
//   MS/MS Instance <-> Device 2 (EL6752)/SolValve
//     PlcTask Outputs/GVL_IO_VALVE.DO_00_V01ChalcogenCarrierChange <-> Connection (Poll)/Outputs/Output Data[0]
//     PlcTask Outputs/GVL_IO_VALVE.DO_00_V02MOCarreirChange <-> Connection (Poll)/Outputs/Output Data[0] @bit 1
//     PlcTask Outputs/GVL_IO_VALVE.DO_00_V03H2SeSourceChange <-> Connection (Poll)/Outputs/Output Data[0] @bit 2
//     PlcTask Outputs/GVL_IO_VALVE.DO_00_V04H2SSourceChange <-> Connection (Poll)/Outputs/Output Data[0] @bit 3
//     PlcTask Outputs/GVL_IO_VALVE.DO_00_V05Source_1TMInCarrierChange <-> Connection (Poll)/Outputs/Output Data[0] @bit 4
//     PlcTask Outputs/GVL_IO_VALVE.DO_00_V06Source_1TMInBypass <-> Connection (Poll)/Outputs/Output Data[0] @bit 5
//     PlcTask Outputs/GVL_IO_VALVE.DO_00_V07Source_2TMGaCarrierChange <-> Connection (Poll)/Outputs/Output Data[0] @bit 6
//     PlcTask Outputs/GVL_IO_VALVE.DO_00_V08Source_2TMGaBypass <-> Connection (Poll)/Outputs/Output Data[0] @bit 7
//     PlcTask Outputs/GVL_IO_VALVE.DO_00_V09Source_3DMSeCarrierChange <-> Connection (Poll)/Outputs/Output Data[1]
//     PlcTask Outputs/GVL_IO_VALVE.DO_00_V10Source_3DMSeBypass <-> Connection (Poll)/Outputs/Output Data[1] @bit 1
//     PlcTask Outputs/GVL_IO_VALVE.DO_00_V11Source_4ChalcogenCarrierChange <-> Connection (Poll)/Outputs/Output Data[1] @bit 2
//     PlcTask Outputs/GVL_IO_VALVE.DO_00_V12Source_4ChalcogenBypass <-> Connection (Poll)/Outputs/Output Data[1] @bit 3
//     PlcTask Outputs/GVL_IO_VALVE.DO_00_V13ReactorPurgeCarrierChange <-> Connection (Poll)/Outputs/Output Data[1] @bit 4
//     PlcTask Outputs/GVL_IO_VALVE.DO_00_V14Source_1TMInManifoldRun <-> Connection (Poll)/Outputs/Output Data[1] @bit 5
//     PlcTask Outputs/GVL_IO_VALVE.DO_00_V15Source_2TMGaManifoldRun <-> Connection (Poll)/Outputs/Output Data[1] @bit 6
//     PlcTask Outputs/GVL_IO_VALVE.DO_00_V16Source_3DMSeManifoldRun <-> Connection (Poll)/Outputs/Output Data[1] @bit 7
//     PlcTask Outputs/GVL_IO_VALVE.DO_00_V17GasH2SeManifoldRun <-> Connection (Poll)/Outputs/Output Data[2]
//     PlcTask Outputs/GVL_IO_VALVE.DO_00_V18GasH2SManifoldRun <-> Connection (Poll)/Outputs/Output Data[2] @bit 1
//     PlcTask Outputs/GVL_IO_VALVE.DO_00_V19Source_4ChalcogenManifoldRun <-> Connection (Poll)/Outputs/Output Data[2] @bit 2
//     PlcTask Outputs/GVL_IO_VALVE.DO_00_V20VentPress_Change <-> Connection (Poll)/Outputs/Output Data[2] @bit 3
//     PlcTask Outputs/GVL_IO_VALVE.DO_00_V21PumpByPass <-> Connection (Poll)/Outputs/Output Data[2] @bit 4
//     PlcTask Outputs/GVL_IO_VALVE.DO_00_V22DORVaccumON <-> Connection (Poll)/Outputs/Output Data[2] @bit 5
//     PlcTask Outputs/GVL_IO_VALVE.DO_00_V23DORFilling <-> Connection (Poll)/Outputs/Output Data[2] @bit 6
//     PlcTask Outputs/GVL_IO_VALVE.DO_00_V24Source_1LeakTest_IN <-> Connection (Poll)/Outputs/Output Data[2] @bit 7
//     PlcTask Outputs/GVL_IO_VALVE.DO_00_V26Source_2LeakTest_IN <-> Connection (Poll)/Outputs/Output Data[3] @bit 1
//     PlcTask Outputs/GVL_IO_VALVE.DO_00_V28Source_3LeakTest_IN <-> Connection (Poll)/Outputs/Output Data[3] @bit 3
//     PlcTask Outputs/GVL_IO_VALVE.DO_00_V30Source_4LeakTest_IN <-> Connection (Poll)/Outputs/Output Data[3] @bit 5
//     PlcTask Outputs/GVL_IO_VALVE.DO_00_V25Source_1LeakTest_OUT <-> Connection (Poll)/Outputs/Output Data[3]
//     PlcTask Outputs/GVL_IO_VALVE.DO_00_V27Source_2LeakTest_OUT <-> Connection (Poll)/Outputs/Output Data[3] @bit 2
//     PlcTask Outputs/GVL_IO_VALVE.DO_00_V29Source_3LeakTest_OUT <-> Connection (Poll)/Outputs/Output Data[3] @bit 4
//     PlcTask Outputs/GVL_IO_VALVE.DO_00_V31Source_4LeakTest_OUT <-> Connection (Poll)/Outputs/Output Data[3] @bit 6
//     PlcTask Outputs/GVL_IO_VALVE.DO_00_V32SourceVacuumON <-> Connection (Poll)/Outputs/Output Data[3] @bit 7
//   MS/MS Instance <-> Device 2 (EL6752)/TempController
//     PlcTask Inputs/GVL_DEVICE_NET_E3508.aInputActiveOut[1] <-> Connection (Poll)/Inputs/Input Data_5
//     PlcTask Inputs/GVL_DEVICE_NET_E3508.aInputActiveOut[2] <-> Connection (Poll)/Inputs/Input Data_6
//     PlcTask Inputs/GVL_DEVICE_NET_E3508.aInputAlarmStatus[1] <-> Connection (Poll)/Inputs/Input Data_7
//     PlcTask Inputs/GVL_DEVICE_NET_E3508.aInputAlarmStatus[2] <-> Connection (Poll)/Inputs/Input Data_8
//     PlcTask Inputs/GVL_DEVICE_NET_E3508.aInputDerivative[1] <-> Connection (Poll)/Inputs/Input Data_17
//     PlcTask Inputs/GVL_DEVICE_NET_E3508.aInputDerivative[2] <-> Connection (Poll)/Inputs/Input Data_18
//     PlcTask Inputs/GVL_DEVICE_NET_E3508.aInputIntegral[1] <-> Connection (Poll)/Inputs/Input Data_15
//     PlcTask Inputs/GVL_DEVICE_NET_E3508.aInputIntegral[2] <-> Connection (Poll)/Inputs/Input Data_16
//     PlcTask Inputs/GVL_DEVICE_NET_E3508.aInputManAutoBytes[1] <-> Connection (Poll)/Inputs/Input Data_9
//     PlcTask Inputs/GVL_DEVICE_NET_E3508.aInputManAutoBytes[2] <-> Connection (Poll)/Inputs/Input Data_10
//     PlcTask Inputs/GVL_DEVICE_NET_E3508.aInputPVBytes[1] <-> Connection (Poll)/Inputs/Input Data_1
//     PlcTask Inputs/GVL_DEVICE_NET_E3508.aInputPVBytes[2] <-> Connection (Poll)/Inputs/Input Data_2
//     PlcTask Inputs/GVL_DEVICE_NET_E3508.aInputProportional[1] <-> Connection (Poll)/Inputs/Input Data_13
//     PlcTask Inputs/GVL_DEVICE_NET_E3508.aInputProportional[2] <-> Connection (Poll)/Inputs/Input Data_14
//     PlcTask Inputs/GVL_DEVICE_NET_E3508.aInputSVBytes[1] <-> Connection (Poll)/Inputs/Input Data_3
//     PlcTask Inputs/GVL_DEVICE_NET_E3508.aInputSVBytes[2] <-> Connection (Poll)/Inputs/Input Data_4
//     PlcTask Inputs/GVL_DEVICE_NET_E3508.aInputStateAutoTune[1] <-> Connection (Poll)/Inputs/Input Data_11
//     PlcTask Inputs/GVL_DEVICE_NET_E3508.aInputStateAutoTune[2] <-> Connection (Poll)/Inputs/Input Data_12
//     PlcTask Outputs/GVL_DEVICE_NET_E3508.aOutputAlarmReset[1] <-> Connection (Poll)/Outputs/Output Data_7
//     PlcTask Outputs/GVL_DEVICE_NET_E3508.aOutputAlarmReset[2] <-> Connection (Poll)/Outputs/Output Data_8
//     PlcTask Outputs/GVL_DEVICE_NET_E3508.aOutputAutoTune_Enable[1] <-> Connection (Poll)/Outputs/Output Data_13
//     PlcTask Outputs/GVL_DEVICE_NET_E3508.aOutputAutoTune_Enable[2] <-> Connection (Poll)/Outputs/Output Data_14
//     PlcTask Outputs/GVL_DEVICE_NET_E3508.aOutputPowerBytes[1] <-> Connection (Poll)/Outputs/Output Data_5
//     PlcTask Outputs/GVL_DEVICE_NET_E3508.aOutputPowerBytes[2] <-> Connection (Poll)/Outputs/Output Data_6
//     PlcTask Outputs/GVL_DEVICE_NET_E3508.aOutputRate[1] <-> Connection (Poll)/Outputs/Output Data_11
//     PlcTask Outputs/GVL_DEVICE_NET_E3508.aOutputRate[2] <-> Connection (Poll)/Outputs/Output Data_12
//     PlcTask Outputs/GVL_DEVICE_NET_E3508.aOutputSVBytes[1] <-> Connection (Poll)/Outputs/Output Data_1
//     PlcTask Outputs/GVL_DEVICE_NET_E3508.aOutputSVBytes[2] <-> Connection (Poll)/Outputs/Output Data_2
//     PlcTask Outputs/GVL_DEVICE_NET_E3508.aOutputThreshold[1] <-> Connection (Poll)/Outputs/Output Data_9
//     PlcTask Outputs/GVL_DEVICE_NET_E3508.aOutputThreshold[2] <-> Connection (Poll)/Outputs/Output Data_10
//     PlcTask Outputs/GVL_DEVICE_NET_E3508.nOutputManAutoBytes[1] <-> Connection (Poll)/Outputs/Output Data_3
//     PlcTask Outputs/GVL_DEVICE_NET_E3508.nOutputManAutoBytes[2] <-> Connection (Poll)/Outputs/Output Data_4
//   MS/MS Instance <-> Device 2 (EL6752)/ThrottleValve
//     PlcTask Inputs/GVL_DEVICE_NET_IQ_PLUS.aInputPressurePV_CDG1[1] <-> Connection (Poll)/Inputs/Input 155_4
//     PlcTask Inputs/GVL_DEVICE_NET_IQ_PLUS.aInputPressurePV_CDG1[2] <-> Connection (Poll)/Inputs/Input 155_5
//     PlcTask Inputs/GVL_DEVICE_NET_IQ_PLUS.aInputPressurePV_CDG2[1] <-> Connection (Poll)/Inputs/Input 155_2
//     PlcTask Inputs/GVL_DEVICE_NET_IQ_PLUS.aInputPressurePV_CDG2[2] <-> Connection (Poll)/Inputs/Input 155_3
//     PlcTask Inputs/GVL_DEVICE_NET_IQ_PLUS.aInputPressureSP[1] <-> Connection (Poll)/Inputs/Input 155_6
//     PlcTask Inputs/GVL_DEVICE_NET_IQ_PLUS.aInputPressureSP[2] <-> Connection (Poll)/Inputs/Input 155_7
//     PlcTask Inputs/GVL_DEVICE_NET_IQ_PLUS.aInputValvePosionPV[1] <-> Connection (Poll)/Inputs/Input 155_8
//     PlcTask Inputs/GVL_DEVICE_NET_IQ_PLUS.aInputValvePosionPV[2] <-> Connection (Poll)/Inputs/Input 155_9
//     PlcTask Inputs/GVL_DEVICE_NET_IQ_PLUS.nInputStatus <-> Connection (Poll)/Inputs/Input 155_1
//     PlcTask Outputs/GVL_DEVICE_NET_IQ_PLUS.aOutputSVBytes[1] <-> Connection (Poll)/Outputs/Output 154[1]
//     PlcTask Outputs/GVL_DEVICE_NET_IQ_PLUS.aOutputSVBytes[2] <-> Connection (Poll)/Outputs/Output 154[2]
//     PlcTask Outputs/GVL_DEVICE_NET_IQ_PLUS.nOutputMode <-> Connection (Poll)/Outputs/Output 154[0]
//     PlcTask Outputs/GVL_DEVICE_NET_IQ_PLUS.nOutputSetType <-> Connection (Poll)/Outputs/Output 154[3]

// ---- DUTs/DUTs/ENUM/E_aAnalogInputIO_Index.TcDUT
{attribute 'qualified_only'}
{attribute 'strict'}
{attribute 'to_string'}
TYPE E_aAnalogInputIO_Index :
(
	E_PV_MFC_01 :=1,
	E_PV_MFC_02 :=2,
	E_PV_MFC_03 :=3,
	E_PV_MFC_04 :=4,
	E_PV_MFC_05 :=5,
	E_PV_MFC_06 :=6,
	E_PV_MFC_07 :=7,
	E_PV_MFC_08 :=8,
	E_PV_MFC_09 :=9,
	E_PV_MFC_10 :=10,
	E_PV_MFC_11 :=11,
	E_PV_MFC_12 :=12,
	E_PV_EPC_01 :=13,
	E_PV_EPC_02 :=14,
	E_PV_EPC_03 :=15,
	E_PV_EPC_04 :=16,
	E_PV_Susceptor_Temp:=17,
	E_PV_Reactor_Pressure:=18,
	E_PV_susceptorRotation:=19
);
END_TYPE

// ---- DUTs/DUTs/ENUM/E_AlarmSetValue.TcDUT
{attribute 'qualified_only'}
{attribute 'strict'}
{attribute 'to_string'}
TYPE E_AlarmSetValue :
(
	E_AS_Alarm_Deviation:=1,
	E_AS_Warning_Deviation,
	E_AS_DelayTime_Analog,
	E_AS_DelayTime_Digital,
	E_AS_Process_Gas_Pressure_Alarm,
	E_AS_Process_Gas_Pressure_Warning,
	E_AS_CWTemp_SH_ALARM,
	E_AS_CWTemp_SH_WARNING,
	E_AS_CWTemp_COIL_ALARM,
	E_AS_CWTemp_COIL_WARNING,
	E_AS_SUSCEPTOR_OVER_TEMP,
	E_AS_REACTOR_OVRE_PRESSURE,
	E_AS_CAN_OPEN_TEMP,
	E_AS_CAN_OPEN_REACTOR_PRESSURE,
	E_AS_DOR_Pressure_Limit,
	E_AS_DOR_RerayCount,
	E_AS_END
);
END_TYPE

// ---- DUTs/DUTs/ENUM/E_Morning_Index.TcDUT
{attribute 'qualified_only'}
{attribute 'strict'}
{attribute 'to_string'}
TYPE E_Morning_Index :
(
	E_Morning_UltimatePressure:=1,
	E_Morning_ExhaustPressure:=2,
	E_Morning_DoubleOring:=3,
	E_Morning_GasPressure_N2:=4,
	E_Morning_GasPressure_H2:=5,
	E_Morning_GasPressure_H2S:=6,
	E_Morning_GasPressure_H2SE:=7,
	E_Morning_CoolingWafer_SH:=8,
	E_Morning_Spare:=9,
	E_Morning_TempPowerRate:=10,
	E_Morning_TV_Position:=11,
	E_Morning_TB_Temp_1:=12,
	E_Morning_TB_Temp_2:=13,
	E_Morning_TB_Temp_3:=14,
	E_Morning_TB_Temp_4:=15,
	E_Morning_Spare16:=16,
	E_Morning_Spare17:=17,
	E_Morning_Total_Flow_MOD:=18,
	E_Morning_Total_Flow_HYD:=19
);
END_TYPE

// ---- DUTs/RecipeStep.TcDUT
TYPE RecipeStep :
STRUCT
	sRecipe : STRING(81);
	iRecipe : ARRAY[1..5] OF INT; //Reactor Condition
	rRecipe : ARRAY[1..30] OF REAL; //MFC, EPC Data
	dRecipe : DWORD; //Valve Data
END_STRUCT
END_TYPE

// ---- GVLs/GVL_CONSTANT.TcGVL
{attribute 'qualified_only'}
VAR_GLOBAL CONSTANT
	EL3064MaxValueH	: REAL := 16383; //0~5V Half Input
	EL3064MaxValue 	: REAL := 32767; //0~10V
	EL4004MaxValueH	: REAL := 16383; //0~5V Half Output
	EL4004MaxValue 	: REAL := 32767; //4~20mA
	EL3102MAxValue	: REAL :=32767;
	
	AnalogControllerOutputVoltage : REAL := 5.0;
	NumAnalogController :UINT:=19;
	NumReactor : UINT := 3;
END_VAR

// ---- GVLs/GVL_DEVICE_NET_E3508.TcGVL
{attribute 'qualified_only'}
VAR_GLOBAL
	(*E3508*)
	(*Input*)
	aInputPVBytes 			AT %I*: ARRAY[1..2]OF USINT; //Loop1 PV
	aInputSVBytes 			AT %I*: ARRAY[1..2]OF USINT; //Loop1 Working PV
	aInputTVBytes 			AT %I*: ARRAY[1..2]OF USINT; //Loop1 Main.TargetSP
	aInputActiveOut 		AT %I*: ARRAY[1..2]OF USINT; //Loop1 Main.ActiveOut
	aInputAlarmStatus 		AT %I*: ARRAY[1..2]OF USINT; //Alarm status
	aInputManAutoBytes 		AT %I*: ARRAY[1..2]OF USINT; // Loop1 Main.AutoMan
	aInputStateAutoTune		AT %I*: ARRAY[1..2]OF USINT; // Loop1 State Auto Tune
	aInputProportional			AT %I*: ARRAY[1..2]OF USINT; // Loop1 State Auto Tune
	aInputIntegral			AT %I*: ARRAY[1..2]OF USINT; // Loop1 State Auto Tune
	aInputDerivative			AT %I*: ARRAY[1..2]OF USINT; // Loop1 State Auto Tune
	
//	aInputAlarmThreshold 	AT %I*: ARRAY[1..2]OF USINT; //Alarm1 Threshold
//	aInputAlarmOut 			AT %I*: ARRAY[1..2]OF USINT; //Alarm.1.Out
//	aInputAlarmSummary 		AT %I*: ARRAY[1..2]OF USINT; // AlmSummary.AnyAlarm (Alarm Clear)

	(*Output*)
	aOutputSVBytes 			AT %Q*: ARRAY[1..2]OF USINT; //Loop.1.Main.TagetSP
	nOutputManAutoBytes 	AT %Q*: ARRAY[1..2]OF USINT; //Loop.1.Main.AutoMan
	aOutputPowerBytes 	AT %Q*: ARRAY[1..2]OF USINT; //Loop1 OP.ManualOutVal
	aOutputAlarmReset	 	AT %Q*: ARRAY[1..2]OF USINT; //Loop1 Alarm Reset
	aOutputThreshold 		AT %Q*: ARRAY[1..2]OF USINT; //Alarm.1.Threshold
	aOutputRate 		AT %Q*: ARRAY[1..2]OF USINT; //Rate
	aOutputAutoTune_Enable 		AT %Q*: ARRAY[1..2]OF USINT; //Auto Tune
	
END_VAR

// ---- GVLs/GVL_IO.TcGVL
{attribute 'qualified_only'}
VAR_GLOBAL
	(* Digital IO to Byte *)
	aDigitalInputIO AT %I* 	: ARRAY[1..9]OF BYTE; //KL1408 9EA
	aDigitalOutputIO AT %Q* : ARRAY[1..5]OF BYTE; //KL2408 4EA
	
	(* Analog Input to INT*)
	aAnalogInputIO AT %I* 	: ARRAY[1..40] OF INT;
	aAnalogOutputIO AT %Q* 	: ARRAY[1..40] OF INT;
	aAnalogInputIO2 AT %I*	: ARRAY[1..2]OF INT;
	
	(*Solenoid Valve*)
	aOutputSolValve AT %Q* 	: DWORD; //Solenoid Valve
	
	aController 			: ARRAY[1..GVL_CONSTANT.NumAnalogController] OF FB_ControlRampGenerator; //MFC, EPC 0 ~ 5V
	aController_PV 			: ARRAY[1..GVL_CONSTANT.NumAnalogController] OF REAL; //Present Value from Device
	aReactorMaxValue		: ARRAY[1..GVL_CONSTANT.NumReactor] OF REAL;
	
	(* Present Value Meter Display*)
	aMonitoring_PV 			: ARRAY[1..16] OF REAL; //Gauge Monitoring Value to UI
	aInputState				: ARRAY[1..6] OF WORD; // Digital Input from Device (Switch)
	aOutputCmd				: ARRAY[1..3] OF WORD; // Digital Command from UI
	aInterlock				: ARRAY[1..5] OF DWORD; // Interlock
	aInterlockSet			: ARRAY[1..20] OF REAL; // UI Interlokc Setting Value
	aInterlockEnable		: ARRAY[1..6] OF DWORD; // UI Interlock Enable Setting
	
	
	nCaseSignalTower		: INT;
	nDorOperationError		: INT;
	bDorState				: BOOL;
	bDorOnEnable			: BOOL;
// 	bE3508_HeaterOn			: BOOL;
	wE3508_CV				: WORD;
	wE3508_PV				: WORD;
	wIqPlus_CV				: WORD;
	wIqPlus_CDG1_PV			: WORD;
	wIqPlus_CDG2_PV			: WORD;
	nRotation_Converted_PV	: REAL;
	rRotation_ControlValue	: REAL;
	nIQPLUS_SetType 		: INT;
	nIQPLUS_Mode			: INT;
	aLineHeater_rTemperaturePV : ARRAY[1..8]OF REAL;
	nE3508_nInputManAutoBytes : USINT;
	isCoverClosed 			: BOOL;
	isPumpRunning 			: BOOL;
	
	UI_INTERLOCK_CHECK_RECIPE_ENABLE:WORD;(**)
	UI_INTERLOCK_CHECK_OPEN_REACTOR:WORD;(**)
END_VAR

// ---- GVLs/GVL.TcGVL
{attribute 'qualified_only'}
VAR_GLOBAL
	MainModule:ST_MAIN_MODULE;
	fbLineHeater_Manager:FB_LINE_HEATER_MANAGER;
	
	RotationResetTon: TON;

END_VAR

// ---- GVLs/GVL_SEQUENCE.TcGVL
{attribute 'qualified_only'}
VAR_GLOBAL
//	fbUpdateModue:FB_UPDATE_MODULE;
	
	fbDeviationCheck		:ARRAY[1..29] OF FB_DeviationCheck;
	fbDeviationCheck_Reactor		:ARRAY[1..3] OF FB_DeviationCheck;
	fbSensorLimitCheck		:ARRAY[1..4] OF FB_SensorLimitCheck;  // Pressure N2 H2 H2S,H2SE 
	fbSensorOverLimitCheck	:ARRAY[1..2] OF FB_OverLimitCheck;  // Over Temp  , Over Pressure  
	fbFaultCheck			:ARRAY[1..8] OF FB_FaultCheck; // CDA/CoolingWafer/Rotation Fault/Vacuum Pump Fault/Gas Cabinet Open / Reactor Door Open / Dor Fault
	fbFaultCheck_Utility	:ARRAY[1..4] OF FB_FaultCheck; //SMPS,Circuit Power , Gas Detector , External Alarm
	fbFaultCheck_Utility_CP :ARRAY[1..4] OF FB_FaultCheck; //CP
END_VAR

// ---- GVLs/GVL_Serial.TcGVL
//{attribute 'qualified_only'}
VAR_GLOBAL
	TxBufferTB : ComBuffer; (* Receive data buffer; used with all receive function blocks *)
	RxBufferTB : ComBuffer; (* Transmit data buffer; used with all receive function blocks *)
	
	TxBufferLH : ComBuffer; //잘동작되면 TB도 지역변수로 변경
	RxBufferLH : ComBuffer;	
END_VAR

// ---- POUs/MAIN.TcPOU
PROGRAM MAIN
VAR_INPUT
	controlModeCmd : E_ControlMode := E_ControlMode.Manual;
END_VAR
VAR
	controlMode	: E_ControlMode := controlModeCmd;
	prevControlMode : E_ControlMode := controlMode;
END_VAR

F_Variable_Valve();
F_Variable_DeviceLink();
F_Variable_FromUI();
F_Variable_FromUI_Interlock();
F_Variable_TODevice();
F_Variable_ToUI_InputState();
GVL.fbLineHeater_Manager(RData_Module_1=>GVL_Serial.LineHeater_data_1,RData_Module_2=>GVL_Serial.LineHeater_data_2);


P11_E3508(); //Temp Controller
P12_IQ_PLUS(); //Throttle Valve Controller
P13_LineHeater();
P14_ThermalBath();
P15_RotationOperation();
P16_CoverOperation();
P17_DOROperation();
P22_Background_ThermalBath();


IF controlMode <> E_ControlMode.Priority THEN
	IF controlMode <> controlModeCmd THEN
		IF controlModeCmd = E_ControlMode.Priority THEN
			prevControlMode := controlMode;
		END_IF
		controlMode := controlModeCmd;
	END_IF
END_IF

CASE controlMode OF
	E_ControlMode.Manual:
		P30_ManualControl();
	
	E_ControlMode.Recipe:
		P50_RecipeControl(); //레시피 콘트론
		
	E_ControlMode.Priority:
		P31_PriorityControl();
		IF P31_PriorityControl.complete = TRUE THEN
			controlMode := prevControlMode;
			controlModeCmd := controlMode;
		END_IF
END_CASE

P70_Interface();
P90_Interlock();
P91_Monitoring();
P92_Maintenance();

END_PROGRAM

// ---- POUs/VARIABLE_LINK/F_Variable_Valve.TcPOU
FUNCTION F_Variable_Valve: BOOL

GVL_IO_VALVE.DO_00_V01ChalcogenCarrierChange :=GVL_IO.aOutputSolValve.0;
GVL_IO_VALVE.DO_00_V02MOCarreirChange :=GVL_IO.aOutputSolValve.1;
GVL_IO_VALVE.DO_00_V03H2SeSourceChange :=GVL_IO.aOutputSolValve.2;
GVL_IO_VALVE.DO_00_V04H2SSourceChange :=GVL_IO.aOutputSolValve.3;
GVL_IO_VALVE.DO_00_V05Source_1TMInCarrierChange :=GVL_IO.aOutputSolValve.4;
GVL_IO_VALVE.DO_00_V06Source_1TMInBypass :=GVL_IO.aOutputSolValve.5;
GVL_IO_VALVE.DO_00_V07Source_2TMGaCarrierChange :=GVL_IO.aOutputSolValve.6;
GVL_IO_VALVE.DO_00_V08Source_2TMGaBypass :=GVL_IO.aOutputSolValve.7;
GVL_IO_VALVE.DO_00_V09Source_3DMSeCarrierChange :=GVL_IO.aOutputSolValve.8;
GVL_IO_VALVE.DO_00_V10Source_3DMSeBypass :=GVL_IO.aOutputSolValve.9;
GVL_IO_VALVE.DO_00_V11Source_4ChalcogenCarrierChange :=GVL_IO.aOutputSolValve.10;
GVL_IO_VALVE.DO_00_V12Source_4ChalcogenBypass :=GVL_IO.aOutputSolValve.11;
GVL_IO_VALVE.DO_00_V13ReactorPurgeCarrierChange :=GVL_IO.aOutputSolValve.12;
GVL_IO_VALVE.DO_00_V14Source_1TMInManifoldRun :=GVL_IO.aOutputSolValve.13;
GVL_IO_VALVE.DO_00_V15Source_2TMGaManifoldRun :=GVL_IO.aOutputSolValve.14;
GVL_IO_VALVE.DO_00_V16Source_3DMSeManifoldRun :=GVL_IO.aOutputSolValve.15;
GVL_IO_VALVE.DO_00_V17GasH2SeManifoldRun :=GVL_IO.aOutputSolValve.16;
GVL_IO_VALVE.DO_00_V18GasH2SManifoldRun :=GVL_IO.aOutputSolValve.17;
GVL_IO_VALVE.DO_00_V19Source_4ChalcogenManifoldRun :=GVL_IO.aOutputSolValve.18;
GVL_IO_VALVE.DO_00_V20VentPress_Change :=GVL_IO.aOutputSolValve.19;
GVL_IO_VALVE.DO_00_V21PumpByPass :=GVL_IO.aOutputSolValve.20;
GVL_IO_VALVE.DO_00_V22DORVaccumON :=GVL_IO.aOutputSolValve.21;
GVL_IO_VALVE.DO_00_V23DORFilling :=GVL_IO.aOutputSolValve.22;
GVL_IO_VALVE.DO_00_V24Source_1LeakTest_IN :=GVL_IO.aOutputSolValve.23;
GVL_IO_VALVE.DO_00_V25Source_1LeakTest_OUT :=GVL_IO.aOutputSolValve.24;
GVL_IO_VALVE.DO_00_V26Source_2LeakTest_IN :=GVL_IO.aOutputSolValve.25;
GVL_IO_VALVE.DO_00_V27Source_2LeakTest_OUT :=GVL_IO.aOutputSolValve.26;
GVL_IO_VALVE.DO_00_V28Source_3LeakTest_IN :=GVL_IO.aOutputSolValve.27;
GVL_IO_VALVE.DO_00_V29Source_3LeakTest_OUT :=GVL_IO.aOutputSolValve.28;
GVL_IO_VALVE.DO_00_V30Source_4LeakTest_IN :=GVL_IO.aOutputSolValve.29;
GVL_IO_VALVE.DO_00_V31Source_4LeakTest_OUT :=GVL_IO.aOutputSolValve.30;
GVL_IO_VALVE.DO_00_V32SourceVacuumON :=GVL_IO.aOutputSolValve.31;

END_FUNCTION

// ---- POUs/VARIABLE_LINK/F_Variable_DeviceLink.TcPOU
FUNCTION F_Variable_DeviceLink: BOOL

GVL_IO.aDigitalInputIO[1].0:=GVL_IO_GAS_CABINET.DI_01_ResetButton ;
GVL_IO.aDigitalInputIO[1].1:=GVL_IO_GAS_CABINET.DI_01_GasCabinetLampButton ;//ok
GVL_IO.aDigitalInputIO[1].2:=GVL_IO_GAS_CABINET.DI_01_PneumaticPressureSensor ;
GVL_IO.aDigitalInputIO[1].3:=GVL_IO_GAS_CABINET.DI_01_GasCabinetDoorClose ;
GVL_IO.aDigitalInputIO[1].4:=GVL_IO_GAS_CABINET.DI_01_ControlCabinetDoorClose ;
GVL_IO.aDigitalInputIO[1].5:=GVL_IO_GAS_CABINET.DI_01_SMPS_1Alarm ;
GVL_IO.aDigitalInputIO[1].6:=GVL_IO_GAS_CABINET.DI_01_SMPS_2Alarm ;
GVL_IO.aDigitalInputIO[1].7:=GVL_IO_GAS_CABINET.DI_01_SMPS_3Alarm ;

GVL_IO.aDigitalInputIO[2].0:=GVL_IO_GAS_CABINET.DI_02_SMPS_4Alarm ;
GVL_IO.aDigitalInputIO[2].1:=GVL_IO_GAS_CABINET.DI_02_GraphiteHeaterELCB ;
GVL_IO.aDigitalInputIO[2].2:=GVL_IO_GAS_CABINET.DI_02_ThermalBathsELCB ;
GVL_IO.aDigitalInputIO[2].3:=GVL_IO_GAS_CABINET.DI_02_VacuumPumpELCB ;
GVL_IO.aDigitalInputIO[2].4:=GVL_IO_GAS_CABINET.DI_02_LineHeatersELCB ;
GVL_IO.aDigitalInputIO[2].5:=GVL_IO_GAS_CABINET.DI_02_RotationMotorCP ;
GVL_IO.aDigitalInputIO[2].6:=GVL_IO_GAS_CABINET.DI_02_CoverLiftMotorCP ;
GVL_IO.aDigitalInputIO[2].7:=GVL_IO_GAS_CABINET.DI_02_T_VCP ;

GVL_IO.aDigitalInputIO[3].0:=GVL_IO_GAS_CABINET.DI_03_GasDetectorCP ;
GVL_IO.aDigitalInputIO[3].1:=GVL_IO_GAS_CABINET.DI_03_CabinetLampsCP ;
GVL_IO.aDigitalInputIO[3].2:=GVL_IO_GAS_CABINET.DI_03_MFCPowerCP ;
GVL_IO.aDigitalInputIO[3].3:=GVL_IO_GAS_CABINET.DI_03_LineHeater_1CP ;
GVL_IO.aDigitalInputIO[3].4:=GVL_IO_GAS_CABINET.DI_03_LineHeater_2CP ;
GVL_IO.aDigitalInputIO[3].5:=GVL_IO_GAS_CABINET.DI_03_LineHeater_3CP ;
GVL_IO.aDigitalInputIO[3].6:=GVL_IO_GAS_CABINET.DI_03_LineHeater_4CP ;
GVL_IO.aDigitalInputIO[3].7:=GVL_IO_GAS_CABINET.DI_03_LineHeater_5CP ;

GVL_IO.aDigitalInputIO[4].0:=GVL_IO_GAS_CABINET.DI_04_LineHeater_6CP ;
GVL_IO.aDigitalInputIO[4].1:=GVL_IO_GAS_CABINET.DI_04_LineHeater_7CP ;
GVL_IO.aDigitalInputIO[4].2:=GVL_IO_GAS_CABINET.DI_04_LineHeater_8CP ;
GVL_IO.aDigitalInputIO[4].3:=GVL_IO_GAS_CABINET.DI_04_GasDetectorH2 ;
GVL_IO.aDigitalInputIO[4].4:=GVL_IO_GAS_CABINET.DI_04_GasDetectorH2S ;
GVL_IO.aDigitalInputIO[4].5:=GVL_IO_GAS_CABINET.DI_04_GasDetectorH2Se ;
GVL_IO.aDigitalInputIO[4].6:=GVL_IO_GAS_CABINET.DI_04_FireSensor ;
GVL_IO.aDigitalInputIO[4].7:=GVL_IO_GAS_CABINET.DI_04_ExternalScrubberFault ;

GVL_IO.aDigitalInputIO[5].0:=GVL_IO_GAS_CABINET.DI_05_ExternalH2GasCabinetFault ;
GVL_IO.aDigitalInputIO[5].1:=GVL_IO_GAS_CABINET.DI_05_ExternalH2SGasCabinetFault ;
GVL_IO.aDigitalInputIO[5].2:=GVL_IO_GAS_CABINET.DI_05_ExternalH2SeGasCabinetFault ;
GVL_IO.aDigitalInputIO[5].3:=GVL_IO_GAS_CABINET.DI_05_ExternalUserInputAlarm ;
GVL_IO.aDigitalInputIO[5].4:=GVL_IO_GAS_CABINET.DI_05_ThermalBath_1DeviationAlarm ;
GVL_IO.aDigitalInputIO[5].5:=GVL_IO_GAS_CABINET.DI_05_ThermalBath_1CutOffAlarm ;
GVL_IO.aDigitalInputIO[5].6:=GVL_IO_GAS_CABINET.DI_05_ThermalBath_2DeviationAlarm ;
GVL_IO.aDigitalInputIO[5].7:=GVL_IO_GAS_CABINET.DI_05_ThermalBath_2CutOffAlarm ;

GVL_IO.aDigitalInputIO[6].0:=GVL_IO_GAS_CABINET.DI_06_ThermalBath_3DeviationAlarm ;
GVL_IO.aDigitalInputIO[6].1:=GVL_IO_GAS_CABINET.DI_06_ThermalBath_3CutOffAlarm ;
GVL_IO.aDigitalInputIO[6].2:=GVL_IO_GAS_CABINET.DI_06_ThermalBath_4DeviationAlarm ;
GVL_IO.aDigitalInputIO[6].3:=GVL_IO_GAS_CABINET.DI_06_ThermalBath_4CutOffAlarm ;
GVL_IO.aDigitalInputIO[6].4:=GVL_IO_GAS_CABINET.DI_06_Spare_01 ;
GVL_IO.aDigitalInputIO[6].5:=GVL_IO_GAS_CABINET.DI_06_Spare_02 ;
GVL_IO.aDigitalInputIO[6].6:=GVL_IO_GAS_CABINET.DI_06_Spare_03 ;
GVL_IO.aDigitalInputIO[6].7:=GVL_IO_GAS_CABINET.DI_06_Spare_04 ;

GVL_IO.aDigitalInputIO[7].0:=GVL_IO_REACTOR_CABINET.DI_01_MaintenanceModeKey ;
GVL_IO.aDigitalInputIO[7].1:=GVL_IO_REACTOR_CABINET.DI_01_ReactorCabinetLampButton ;
GVL_IO.aDigitalInputIO[7].2:=GVL_IO_REACTOR_CABINET.DI_01_DORVACButton ; //Sheet에서는 빠짐
GVL_IO.aDigitalInputIO[7].3:=GVL_IO_REACTOR_CABINET.DI_01_DORATMButton ;//Sheet에서는 빠짐
GVL_IO.aDigitalInputIO[7].4:=GVL_IO_REACTOR_CABINET.DI_01_ReactorDoorUpButton ;//Sheet에서는 빠짐
GVL_IO.aDigitalInputIO[7].5:=GVL_IO_REACTOR_CABINET.DI_01_ReactorDoorDownButton ;//Sheet에서는 빠짐
GVL_IO.aDigitalInputIO[7].6:=GVL_IO_REACTOR_CABINET.DI_01_ClampLock ;//Sheet에서는 빠짐
GVL_IO.aDigitalInputIO[7].7:=GVL_IO_REACTOR_CABINET.DI_01_ClampRelease ;//Sheet에서는 빠짐

GVL_IO.aDigitalInputIO[8].0:=GVL_IO_REACTOR_CABINET.DI_02_C_WFlowSensor ;
GVL_IO.aDigitalInputIO[8].1:=GVL_IO_REACTOR_CABINET.DI_02_SusceptorRotationMotorFault ;
GVL_IO.aDigitalInputIO[8].2:=GVL_IO_REACTOR_CABINET.DI_02_VacuumPumpFail ;
GVL_IO.aDigitalInputIO[8].3:=GVL_IO_REACTOR_CABINET.DI_02_VacuumPumpWarning ;
GVL_IO.aDigitalInputIO[8].4:=GVL_IO_REACTOR_CABINET.DI_02_VacuumPumpAlarm ;
GVL_IO.aDigitalInputIO[8].5:=GVL_IO_REACTOR_CABINET.DI_02_VacuumPumpFBRunning ;
GVL_IO.aDigitalInputIO[8].6:=GVL_IO_REACTOR_CABINET.DI_02_VacuumPumpRunning ;
GVL_IO.aDigitalInputIO[8].7:=GVL_IO_REACTOR_CABINET.DI_02_ReactorDoorUpLimitSensor ;

GVL_IO.aDigitalInputIO[9].0:=GVL_IO_REACTOR_CABINET.DI_03_ReactorDoorDownLimitSensor ;
GVL_IO.aDigitalInputIO[9].1:=GVL_IO_REACTOR_CABINET.DI_03_CylinderAutoSwitch_Closed ;
GVL_IO.aDigitalInputIO[9].2:=GVL_IO_REACTOR_CABINET.DI_03_CylinderAutoSwitch_Opened ;
GVL_IO.aDigitalInputIO[9].3:=GVL_IO_REACTOR_CABINET.DI_03_ReactorCabinetDoorClose ;
GVL_IO.aDigitalInputIO[9].4:=GVL_IO_REACTOR_CABINET.DI_03_Spare_01 ;
GVL_IO.aDigitalInputIO[9].5:=GVL_IO_REACTOR_CABINET.DI_03_Spare_02 ;
GVL_IO.aDigitalInputIO[9].6:=GVL_IO_REACTOR_CABINET.DI_03_Spare_03 ;
GVL_IO.aDigitalInputIO[9].7:=GVL_IO_REACTOR_CABINET.DI_03_Spare_04 ;


GVL_IO.aDigitalOutputIO[1].0:=GVL_IO_GAS_CABINET.DO_07_SystemPowerOffLock ; //Sheet에서는 빠짐
GVL_IO.aDigitalOutputIO[1].1:=GVL_IO_GAS_CABINET.DO_07_ControlCabinetLamp ;//Sheet에서는 빠짐
GVL_IO.aDigitalOutputIO[1].2:=GVL_IO_GAS_CABINET.DO_07_GasCabinetLamp ;//Sheet에서는 빠짐
GVL_IO.aDigitalOutputIO[1].3:=GVL_IO_GAS_CABINET.DO_07_GraphiteHeaterMC ;//Sheet에서는 빠짐
GVL_IO.aDigitalOutputIO[1].4:=GVL_IO_GAS_CABINET.DO_07_ThermalBathsMC ;//Sheet에서는 빠짐
GVL_IO.aDigitalOutputIO[1].5:=GVL_IO_GAS_CABINET.DO_07_VacuumPumpMC ;//Sheet에서는 빠짐
GVL_IO.aDigitalOutputIO[1].6:=GVL_IO_GAS_CABINET.DO_07_LineHeatersMC ;//Sheet에서는 빠짐
GVL_IO.aDigitalOutputIO[1].7:=GVL_IO_GAS_CABINET.DO_07_ResetButtonLamp ;//Sheet에서는 빠짐

GVL_IO.aDigitalOutputIO[2].0:=GVL_IO_GAS_CABINET.DO_08_Spare_01 ;
GVL_IO.aDigitalOutputIO[2].1:=GVL_IO_GAS_CABINET.DO_08_Spare_02 ;
GVL_IO.aDigitalOutputIO[2].2:=GVL_IO_GAS_CABINET.DO_08_Spare_03 ;
GVL_IO.aDigitalOutputIO[2].3:=GVL_IO_GAS_CABINET.DO_08_Spare_04 ;
GVL_IO.aDigitalOutputIO[2].4:=GVL_IO_GAS_CABINET.DO_08_Spare_05 ;
GVL_IO.aDigitalOutputIO[2].5:=GVL_IO_GAS_CABINET.DO_08_Spare_06 ;
GVL_IO.aDigitalOutputIO[2].6:=GVL_IO_GAS_CABINET.DO_08_Spare_07 ;
GVL_IO.aDigitalOutputIO[2].7:=GVL_IO_GAS_CABINET.DO_08_Spare_08 ;

GVL_IO.aDigitalOutputIO[3].0:=GVL_IO_REACTOR_CABINET.DO_04_SignalTowerRed ;
GVL_IO.aDigitalOutputIO[3].1:=GVL_IO_REACTOR_CABINET.DO_04_SignalTowerOrange ;
GVL_IO.aDigitalOutputIO[3].2:=GVL_IO_REACTOR_CABINET.DO_04_SignalTowerGreen ;
GVL_IO.aDigitalOutputIO[3].3:=GVL_IO_REACTOR_CABINET.DO_04_SignalTowerBlue ;
GVL_IO.aDigitalOutputIO[3].4:=GVL_IO_REACTOR_CABINET.DO_04_SignalTowerWhite ;
GVL_IO.aDigitalOutputIO[3].5:=GVL_IO_REACTOR_CABINET.DO_04_SignalTowerBuzzer ;
GVL_IO.aDigitalOutputIO[3].6:=GVL_IO_REACTOR_CABINET.DO_04_ReactorCoverUpRelay ; //Sheet에서는 빠짐
GVL_IO.aDigitalOutputIO[3].7:=GVL_IO_REACTOR_CABINET.DO_04_ReactorCoverDownRelay ;//Sheet에서는 빠짐

GVL_IO.aDigitalOutputIO[4].0:=GVL_IO_REACTOR_CABINET.DO_05_ClampLock ;
GVL_IO.aDigitalOutputIO[4].1:=GVL_IO_REACTOR_CABINET.DO_05_ClampRelease ;
GVL_IO.aDigitalOutputIO[4].2:=GVL_IO_REACTOR_CABINET.DO_05_VacuumPumpStart_Stop ;//Sheet에서는 빠짐
GVL_IO.aDigitalOutputIO[4].3:=GVL_IO_REACTOR_CABINET.DO_05_VacuumPumpReset ;//Sheet에서는 빠짐
GVL_IO.aDigitalOutputIO[4].4:=GVL_IO_REACTOR_CABINET.DO_05_SusceptorRotationFWD ;
GVL_IO.aDigitalOutputIO[4].5:=GVL_IO_REACTOR_CABINET.DO_05_SusceptorRotationSTOP ;
GVL_IO.aDigitalOutputIO[4].6:=GVL_IO_REACTOR_CABINET.DO_05_SusceptorRotationAL_RST ;//Sheet에서는 빠짐
GVL_IO.aDigitalOutputIO[4].7:=GVL_IO_REACTOR_CABINET.DO_05_DORVACButtonLamp ;//Sheet에서는 빠짐

GVL_IO.aDigitalOutputIO[5].0:=GVL_IO_REACTOR_CABINET.DO_06_DORATMButtonLamp ;//Sheet에서는 빠짐
GVL_IO.aDigitalOutputIO[5].1:=GVL_IO_REACTOR_CABINET.DO_06_ReactorCoverUpButtonLamp ;//Sheet에서는 빠짐
GVL_IO.aDigitalOutputIO[5].2:=GVL_IO_REACTOR_CABINET.DO_06_ReactorCoverDownButtonLamp ;//Sheet에서는 빠짐
GVL_IO.aDigitalOutputIO[5].3:=GVL_IO_REACTOR_CABINET.DO_06_ClampLockButtonLamp ;//Sheet에서는 빠짐
GVL_IO.aDigitalOutputIO[5].4:=GVL_IO_REACTOR_CABINET.DO_06_ClampReleaseButtonLamp ;//Sheet에서는 빠짐
GVL_IO.aDigitalOutputIO[5].5:=GVL_IO_REACTOR_CABINET.DO_06_ReactorCabinetLamp ;//Sheet에서는 빠짐
GVL_IO.aDigitalOutputIO[5].6:=GVL_IO_REACTOR_CABINET.DO_06_Spare07 ;//Sheet에서는 빠짐
GVL_IO.aDigitalOutputIO[5].7:=GVL_IO_REACTOR_CABINET.DO_06_Spare08 ;//Sheet에서는 빠짐


GVL_IO.aAnalogInputIO[1]:=GVL_IO_GAS_CABINET.AI_09_M01_ChalcogenRunPV ;
GVL_IO.aAnalogInputIO[2]:=GVL_IO_GAS_CABINET.AI_09_M02_MORunPV ;
GVL_IO.aAnalogInputIO[3]:=GVL_IO_GAS_CABINET.AI_09_M03_H2SeSupplyPV ;
GVL_IO.aAnalogInputIO[4]:=GVL_IO_GAS_CABINET.AI_09_M04_H2SSupplyPV ;
GVL_IO.aAnalogInputIO[5]:=GVL_IO_GAS_CABINET.AI_11_M05_Source_1TMInSupplyPV ;
GVL_IO.aAnalogInputIO[6]:=GVL_IO_GAS_CABINET.AI_11_M06_Source_2TMGaSupplyPV ;
GVL_IO.aAnalogInputIO[7]:=GVL_IO_GAS_CABINET.AI_11_M07_Source_3DMSeSupplyPV ;
GVL_IO.aAnalogInputIO[8]:=GVL_IO_GAS_CABINET.AI_11_M08_Source_4ChalcoSupplyPV ;
GVL_IO.aAnalogInputIO[9]:=GVL_IO_GAS_CABINET.AI_13_M09_LinerPurgePV ;
GVL_IO.aAnalogInputIO[10]:=GVL_IO_GAS_CABINET.AI_13_M10_HeaterPurgePV ;
GVL_IO.aAnalogInputIO[11]:=GVL_IO_GAS_CABINET.AI_13_M11_ChalcogenVentPV ;
GVL_IO.aAnalogInputIO[12]:=GVL_IO_GAS_CABINET.AI_13_M12_MOVentPV ;
GVL_IO.aAnalogInputIO[13]:=GVL_IO_GAS_CABINET.AI_15_E01Source_1TMInPressurePV ;
GVL_IO.aAnalogInputIO[14]:=GVL_IO_GAS_CABINET.AI_15_E02Source_2TMGaPressurePV ;
GVL_IO.aAnalogInputIO[15]:=GVL_IO_GAS_CABINET.AI_15_E03Source_3DMSePressurePV ;
GVL_IO.aAnalogInputIO[16]:=GVL_IO_GAS_CABINET.AI_15_E04Source_4ChalcoPressurePV ;

GVL_IO.aAnalogInputIO[19]:=GVL_IO_REACTOR_CABINET.AI_08_R01SusceptorRotationPV ;
GVL_IO.aAnalogInputIO[20]:=GVL_IO_REACTOR_CABINET.AI_07_P02_ReactorPressure10TorrPV;
GVL_IO.aAnalogInputIO[21]:=GVL_IO_REACTOR_CABINET.AI_07_P03_ExhaustPressurePV ;
GVL_IO.aAnalogInputIO[22]:=GVL_IO_REACTOR_CABINET.AI_07_S05_DORPressurePV ;

GVL_IO.aAnalogInputIO[23]:=GVL_IO_GAS_CABINET.DI_18_S01N2SupplyPressPV ;
GVL_IO.aAnalogInputIO[24]:=GVL_IO_GAS_CABINET.DI_18_S02H2SupplyPressPV ;
GVL_IO.aAnalogInputIO[25]:=GVL_IO_GAS_CABINET.DI_18_S03H2SSupplyPressPV ;
GVL_IO.aAnalogInputIO[26]:=GVL_IO_GAS_CABINET.DI_18_S04H2SeSupplyPressPV ;
GVL_IO.aAnalogInputIO[27]:=GVL_IO_REACTOR_CABINET.AI_10_R04S_HCoolingWaterPV ;


GVL_IO.aAnalogInputIO2[1]:=GVL_IO_GAS_CABINET.DI_17_DP1ChalcogenDP ;
GVL_IO.aAnalogInputIO2[2]:=GVL_IO_GAS_CABINET.DI_17_DP2MODP ;


//GVL_IO.aAnalogInputIO[24]:=GVL_IO_REACTOR_CABINET.AI_07_Spare_04 ;
//GVL_IO.aAnalogInputIO[26]:=GVL_IO_REACTOR_CABINET.AI_08_Spare_02 ;
//GVL_IO.aAnalogInputIO[27]:=GVL_IO_REACTOR_CABINET.AI_08_Spare_03 ;
//GVL_IO.aAnalogInputIO[28]:=GVL_IO_REACTOR_CABINET.AI_08_Spare_04 ;


//GVL_IO.aAnalogInputIO[30]:=GVL_IO_REACTOR_CABINET.AI_10_Spare_02 ;
//GVL_IO.aAnalogInputIO[31]:=GVL_IO_REACTOR_CABINET.AI_10_Spare_03 ;
//GVL_IO.aAnalogInputIO[32]:=GVL_IO_REACTOR_CABINET.AI_10_Spare_04 ;


GVL_IO_GAS_CABINET.AO_10_M01_ChalcogenRunSV :=GVL_IO.aAnalogOutputIO[1];
GVL_IO_GAS_CABINET.AO_10_M02_MORunSV :=GVL_IO.aAnalogOutputIO[2];
GVL_IO_GAS_CABINET.AO_10_M03_H2SeSupplySV  := GVL_IO.aAnalogOutputIO[3];
GVL_IO_GAS_CABINET.AO_10_M04_H2SSupplySV :=GVL_IO.aAnalogOutputIO[4];

GVL_IO_GAS_CABINET.AO_12_M05_Source_1TMInSupplySV :=GVL_IO.aAnalogOutputIO[5];
GVL_IO_GAS_CABINET.AO_12_M06_Source_2TMGaSupplySV :=GVL_IO.aAnalogOutputIO[6];
GVL_IO_GAS_CABINET.AO_12_M07_Source_3DMSeSupplySV :=GVL_IO.aAnalogOutputIO[7];
GVL_IO_GAS_CABINET.AO_12_M08_Source_4ChalcoSupplySV :=GVL_IO.aAnalogOutputIO[8];
GVL_IO_GAS_CABINET.AO_14_M09_LinerPurgeSV :=GVL_IO.aAnalogOutputIO[9];
GVL_IO_GAS_CABINET.AO_14_M10_HeaterPurgeSV :=GVL_IO.aAnalogOutputIO[10];
GVL_IO_GAS_CABINET.AO_14_M11_ChalcogenVentSV :=GVL_IO.aAnalogOutputIO[11];
GVL_IO_GAS_CABINET.AO_14_M12_MOVentSV :=GVL_IO.aAnalogOutputIO[12];
GVL_IO_GAS_CABINET.AO_16_E01Source_1TMInPressureSV :=GVL_IO.aAnalogOutputIO[13];
GVL_IO_GAS_CABINET.AO_16_E02Source_2TMGaPressureSV :=GVL_IO.aAnalogOutputIO[14];
GVL_IO_GAS_CABINET.AO_16_E03Source_3DMSePressureSV :=GVL_IO.aAnalogOutputIO[15];
GVL_IO_GAS_CABINET.AO_16_E04Source_4ChalcoPressureSV :=GVL_IO.aAnalogOutputIO[16];

//GVL_IO_REACTOR_CABINET.AO_09_P03_ExhaustPressureAM215Input:=GVL_IO.aAnalogOutputIO[17];

GVL_IO_REACTOR_CABINET.AO_09_P03_ExhaustPressureAM215Input:=GVL_IO_REACTOR_CABINET.AI_07_P03_ExhaustPressurePV;


GVL_IO_REACTOR_CABINET.AO_09_R01_SusceptorRotationSV:=GVL_IO.aAnalogOutputIO[18];
GVL_IO_REACTOR_CABINET.AO_09_Spare_03:=GVL_IO.aAnalogOutputIO[19];
GVL_IO_REACTOR_CABINET.AO_09_Spare_04 :=GVL_IO.aAnalogOutputIO[20];

END_FUNCTION

// ---- POUs/VARIABLE_LINK/F_Variable_FromUI.TcPOU
FUNCTION F_Variable_FromUI: BOOL


VAR
	rRotationAlarm_Reset: R_TRIG;
	
	Rotation_Shift: WORD;
END_VAR

////UI에서 Write하는 Command
//아래 MC는 Maint 모드에서만 조작 가능
//GVL_COMMAND_FROM_UI.CMD_HEATER_MAIN_MC_ON:= GVL_IO.aOutputCmd[1].0;
//GVL_COMMAND_FROM_UI.CMD_THERMAL_BACH_MC_ON:= GVL_IO.aOutputCmd[1].1;
//GVL_COMMAND_FROM_UI.CMD_VACUUM_PUMP_MC_ON:= GVL_IO.aOutputCmd[1].2;
//GVL_COMMAND_FROM_UI.CMD_LINE_HEATER_MC_ON := GVL_IO.aOutputCmd[1].3;

GVL_COMMAND_FROM_UI.CMD_VACUUM_PUMP_ON := GVL_IO.aOutputCmd[1].6;
GVL_COMMAND_FROM_UI.CMD_VACUUM_PUMP_RESET:= GVL_IO.aOutputCmd[1].7;

GVL_COMMAND_FROM_UI.CMD_ROTATION_START:= GVL_IO.aOutputCmd[1].8;
GVL_COMMAND_FROM_UI.CMD_ROTATION_RESET := GVL_IO.aOutputCmd[1].10;

//jhkang 하드웨어로 구성 되어 있어야 하는데 아직 구성 안됨 := GVL_IO.aOutputCmd[1].10;
GVL_COMMAND_FROM_UI.CMD_E3508_MAN_AUTO := GVL_IO.aOutputCmd[1].12;(*True:Manual  False:auto*)
GVL_COMMAND_FROM_UI.CMD_THROTTLE_PRESSURE_POSITION_MODE := GVL_IO.aOutputCmd[1].13;//true: Pressure False:Position

GVL_COMMAND_FROM_UI.CMD_THROTTLE_OUTPUT_MODE:= WORD_TO_USINT(GVL_IO.aOutputCmd[2]); //Throttle Valve Mode Setting 0:Normal 1:Close 2:Open 3:Hold 4:Reset

GVL_IO_GAS_CABINET.DO_07_GraphiteHeaterMC :=  GVL_COMMAND_FROM_UI.CMD_HEATER_MAIN_MC_ON;
GVL_IO_GAS_CABINET.DO_07_ThermalBathsMC :=  GVL_COMMAND_FROM_UI.CMD_THERMAL_BACH_MC_ON;
GVL_IO_GAS_CABINET.DO_07_VacuumPumpMC :=  GVL_COMMAND_FROM_UI.CMD_VACUUM_PUMP_MC_ON;
GVL_IO_GAS_CABINET.DO_07_LineHeatersMC:=  GVL_COMMAND_FROM_UI.CMD_LINE_HEATER_MC_ON;

GVL_IO_REACTOR_CABINET.DO_05_SusceptorRotationFWD:=GVL_COMMAND_FROM_UI.CMD_ROTATION_START;

rRotationAlarm_Reset(CLK:=GVL_COMMAND_FROM_UI.CMD_ROTATION_RESET);
IF rRotationAlarm_Reset.Q THEN
	GVL_IO_REACTOR_CABINET.DO_05_SusceptorRotationAL_RST:=TRUE;
END_IF

GVL.RotationResetTon(IN:=GVL_IO_REACTOR_CABINET.DO_05_SusceptorRotationAL_RST,PT:=T#3S);

IF GVL_IO_REACTOR_CABINET.DI_02_SusceptorRotationMotorFault = TRUE OR GVL.RotationResetTon.Q THEN
	GVL.RotationResetTon(in:=FALSE);
	IF GVL_IO_REACTOR_CABINET.DO_05_SusceptorRotationAL_RST = TRUE THEN
		GVL_IO_REACTOR_CABINET.DO_05_SusceptorRotationAL_RST:=FALSE;
	END_IF
	
	IF GVL_IO.aOutputCmd[1].10 = TRUE THEN
		GVL_IO.aOutputCmd[1].10:=FALSE;
	END_IF
END_IF


	//GVL_IO_REACTOR_CABINET.DO_05_SusceptorRotationAL_RST:=GVL_COMMAND_FROM_UI.CMD_ROTATION_RESET;	
GVL_IO_REACTOR_CABINET.DO_05_VacuumPumpStart_Stop := GVL_COMMAND_FROM_UI.CMD_VACUUM_PUMP_ON;
GVL_IO_REACTOR_CABINET.DO_05_VacuumPumpReset:=GVL_COMMAND_FROM_UI.CMD_VACUUM_PUMP_RESET;

END_FUNCTION

// ---- POUs/VARIABLE_LINK/F_Variable_FromUI_Interlock.TcPOU
FUNCTION F_Variable_FromUI_Interlock: BOOL

END_FUNCTION

// ---- POUs/VARIABLE_LINK/F_Variable_ToUI_InputState.TcPOU
FUNCTION F_Variable_ToUI_InputState: BOOL

VAR
	Cout: INT;
END_VAR

(* UI Right Dashboard Variable*)
GVL_IO.aInputState[1].0 := GVL_IO_REACTOR_CABINET.DI_01_MaintenanceModeKey; //Maintenance Key
GVL_IO.aInputState[1].1	:= GVL_IO_REACTOR_CABINET.DO_06_ReactorCabinetLamp; //Reactor Cabinet Lamp
GVL_IO.aInputState[1].2	:= GVL_IO_GAS_CABINET.DO_07_GasCabinetLamp; // Gas Cabinet Lamp
GVL_IO.aInputState[1].3	:= GVL_IO_GAS_CABINET.DI_01_PneumaticPressureSensor; // Power Cabinet Lamp
GVL_IO.aInputState[1].4 := GVL_IO_REACTOR_CABINET.DI_02_C_WFlowSensor; //CDA Alarm Switch
GVL_IO.aInputState[1].5	:=GVL_IO_REACTOR_CABINET.DO_05_SusceptorRotationFWD;

IF GVL_IO_REACTOR_CABINET.DO_05_SusceptorRotationFWD = FALSE THEN
	Cout:=Cout+1;
END_IF
GVL_IO.aInputState[1].6 :=GVL_IO_REACTOR_CABINET.DO_05_SusceptorRotationSTOP; 
GVL_IO.aInputState[1].7 :=NOT GVL_IO_REACTOR_CABINET.DI_02_SusceptorRotationMotorFault; //Susceptor Rotation Motor
GVL_IO.aInputState[1].8 := GVL_IO_REACTOR_CABINET.DI_02_VacuumPumpFail; //Vacuum Pump
GVL_IO.aInputState[1].9 := GVL_IO_REACTOR_CABINET.DI_02_VacuumPumpWarning; //Vacuum Pump
GVL_IO.aInputState[1].10 := GVL_IO_REACTOR_CABINET.DI_02_VacuumPumpAlarm; //Vacuum Pump
GVL_IO.aInputState[1].11 := GVL_IO_REACTOR_CABINET.DI_02_VacuumPumpFBRunning; //Vacuum Pump
GVL_IO.aInputState[1].12 := GVL_IO_REACTOR_CABINET.DI_02_VacuumPumpFBRunning; //Vacuum Pump

GVL_IO.aInputState[1].13 := GVL_IO_REACTOR_CABINET.DI_03_ReactorCabinetDoorClose;
GVL_IO.aInputState[1].14 := GVL_IO_GAS_CABINET.DI_01_GasCabinetDoorClose;
GVL_IO.aInputState[1].15 := GVL_IO_GAS_CABINET.DI_01_ControlCabinetDoorClose;

GVL_IO.aInputState[2].0	:= GVL_IO_GAS_CABINET.DI_01_ResetButton;
GVL_IO.aInputState[2].1	:= GVL_IO_REACTOR_CABINET.DI_02_ReactorDoorUpLimitSensor;
GVL_IO.aInputState[2].2	:= GVL_IO_REACTOR_CABINET.DI_03_ReactorDoorDownLimitSensor;
GVL_IO.aInputState[2].3	:= GVL_IO_REACTOR_CABINET.DI_03_CylinderAutoSwitch_Closed;
GVL_IO.aInputState[2].4	:= GVL_IO_REACTOR_CABINET.DI_03_CylinderAutoSwitch_Opened;
GVL_IO.aInputState[2].5	:= NOT GVL_IO_GAS_CABINET.DI_01_SMPS_1Alarm;
GVL_IO.aInputState[2].6	:= NOT GVL_IO_GAS_CABINET.DI_01_SMPS_2Alarm;
GVL_IO.aInputState[2].7	:= NOT GVL_IO_GAS_CABINET.DI_01_SMPS_3Alarm;
GVL_IO.aInputState[2].8	:= NOT GVL_IO_GAS_CABINET.DI_02_SMPS_4Alarm;
GVL_IO.aInputState[2].9	:= GVL_IO_GAS_CABINET.DI_02_GraphiteHeaterELCB;
GVL_IO.aInputState[2].10:= GVL_IO_GAS_CABINET.DI_02_ThermalBathsELCB;
GVL_IO.aInputState[2].11:= GVL_IO_GAS_CABINET.DI_02_VacuumPumpELCB;
GVL_IO.aInputState[2].12:= GVL_IO_GAS_CABINET.DI_02_LineHeatersELCB;
GVL_IO.aInputState[2].13:= GVL_IO_GAS_CABINET.DI_02_RotationMotorCP;
GVL_IO.aInputState[2].14:= GVL_IO_GAS_CABINET.DI_02_CoverLiftMotorCP;
GVL_IO.aInputState[2].15:= GVL_IO_GAS_CABINET.DI_02_T_VCP;

GVL_IO.aInputState[3].0:= GVL_IO_GAS_CABINET.DI_03_GasDetectorCP;
GVL_IO.aInputState[3].1:= GVL_IO_GAS_CABINET.DI_03_CabinetLampsCP;
GVL_IO.aInputState[3].2:= GVL_IO_GAS_CABINET.DI_03_MFCPowerCP;
GVL_IO.aInputState[3].3:= GVL_IO_GAS_CABINET.DI_03_LineHeater_1CP;
GVL_IO.aInputState[3].4:= GVL_IO_GAS_CABINET.DI_03_LineHeater_2CP;
GVL_IO.aInputState[3].5:= GVL_IO_GAS_CABINET.DI_03_LineHeater_3CP;
GVL_IO.aInputState[3].6:= GVL_IO_GAS_CABINET.DI_03_LineHeater_4CP;
GVL_IO.aInputState[3].7:= GVL_IO_GAS_CABINET.DI_03_LineHeater_5CP;
GVL_IO.aInputState[3].8:= GVL_IO_GAS_CABINET.DI_04_LineHeater_6CP;
GVL_IO.aInputState[3].9:= GVL_IO_GAS_CABINET.DI_04_LineHeater_7CP;
GVL_IO.aInputState[3].10:= GVL_IO_GAS_CABINET.DI_04_LineHeater_8CP;

GVL_IO.aInputState[3].11:= GVL_IO_GAS_CABINET.DI_04_GasDetectorH2;
GVL_IO.aInputState[3].12:= GVL_IO_GAS_CABINET.DI_04_GasDetectorH2S;
GVL_IO.aInputState[3].13:= GVL_IO_GAS_CABINET.DI_04_GasDetectorH2Se;
GVL_IO.aInputState[3].14:= GVL_IO_GAS_CABINET.DI_04_FireSensor;
GVL_IO.aInputState[3].15 := GVL_IO_GAS_CABINET.DI_04_ExternalScrubberFault;

GVL_IO.aInputState[4].0 := GVL_IO_GAS_CABINET.DI_05_ExternalH2GasCabinetFault;
GVL_IO.aInputState[4].1 := GVL_IO_GAS_CABINET.DI_05_ExternalH2SGasCabinetFault;
GVL_IO.aInputState[4].2 := GVL_IO_GAS_CABINET.DI_05_ExternalH2SeGasCabinetFault;
GVL_IO.aInputState[4].3 := GVL_IO_GAS_CABINET.DI_05_ExternalUserInputAlarm;

GVL_IO.aInputState[4].4:= GVL_IO_GAS_CABINET.DI_05_ThermalBath_1DeviationAlarm;
GVL_IO.aInputState[4].5:= GVL_IO_GAS_CABINET.DI_05_ThermalBath_1CutOffAlarm;
GVL_IO.aInputState[4].6:= GVL_IO_GAS_CABINET.DI_05_ThermalBath_2DeviationAlarm;
GVL_IO.aInputState[4].7:= GVL_IO_GAS_CABINET.DI_05_ThermalBath_2CutOffAlarm;
GVL_IO.aInputState[4].8:= GVL_IO_GAS_CABINET.DI_06_ThermalBath_3DeviationAlarm;
GVL_IO.aInputState[4].9:= GVL_IO_GAS_CABINET.DI_06_ThermalBath_3CutOffAlarm;
GVL_IO.aInputState[4].10:= GVL_IO_GAS_CABINET.DI_06_ThermalBath_4DeviationAlarm;
GVL_IO.aInputState[4].11:= GVL_IO_GAS_CABINET.DI_06_ThermalBath_3CutOffAlarm;


GVL_IO.aInputState[5].0:= GVL_IO_REACTOR_CABINET.DO_04_SignalTowerRed;
GVL_IO.aInputState[5].1:= GVL_IO_REACTOR_CABINET.DO_04_SignalTowerOrange;
GVL_IO.aInputState[5].2:= GVL_IO_REACTOR_CABINET.DO_04_SignalTowerGreen;
GVL_IO.aInputState[5].3:= GVL_IO_REACTOR_CABINET.DO_04_SignalTowerBlue;
GVL_IO.aInputState[5].4:= GVL_IO_REACTOR_CABINET.DO_04_SignalTowerWhite;
GVL_IO.aInputState[5].5:= GVL_IO_REACTOR_CABINET.DO_04_SignalTowerBuzzer;

GVL_IO.aInputState[5].6:= GVL_IO_REACTOR_CABINET.DI_01_ClampLock;
GVL_IO.aInputState[5].7:= GVL_IO_REACTOR_CABINET.DI_01_ClampRelease;

GVL_IO.aInputState[5].8:= F_GetDorPressure(GVL_IO_REACTOR_CABINET.AI_07_S05_DORPressurePV) < 100;
GVL_IO.aInputState[5].9:= GVL_DEVICE_NET_E3508.aInputAlarmStatus[1] > 0 OR GVL_DEVICE_NET_E3508.aInputAlarmStatus[2] > 0 ;
GVL_IO.aInputState[5].10:= GVL_DEVICE_NET_E3508.aInputManAutoBytes[1].0;//(*True:manual   False:auto*)

GVL_IO.aInputState[6].0:= GVL_DEVICE_NET_IQ_PLUS.nInputStatus  = 0;
GVL_IO.aInputState[6].1:= GVL_DEVICE_NET_IQ_PLUS.nInputStatus  = 1;
GVL_IO.aInputState[6].2:= GVL_DEVICE_NET_IQ_PLUS.nInputStatus  = 2;
GVL_IO.aInputState[6].3:= GVL_DEVICE_NET_IQ_PLUS.nInputStatus  = 3;
GVL_IO.aInputState[6].4:= GVL_DEVICE_NET_IQ_PLUS.nInputStatus  = 4;
GVL_IO.aInputState[6].5:= GVL_DEVICE_NET_IQ_PLUS.nInputStatus  = 5;
GVL_IO.aInputState[6].6:= GVL_DEVICE_NET_IQ_PLUS.nInputStatus  = 6;
GVL_IO.aInputState[6].7:= GVL_DEVICE_NET_IQ_PLUS.nInputStatus  = 7;
GVL_IO.aInputState[6].8:= GVL_DEVICE_NET_IQ_PLUS.nInputStatus  = 8;

GVL_IO.aInputState[6].9:= P90_Interlock.bRecipeStartAvailable;
GVL_IO.aInputState[6].10:= P90_Interlock.bReactorOpenEnable;
GVL_IO.aInputState[6].12:= GVL_IO_REACTOR_CABINET.DI_03_ReactorDoorDownLimitSensor AND P90_Interlock.AlarmTrig = FALSE AND GVL_IO_VALVE.DO_00_V21PumpByPass = FALSE;

END_FUNCTION

// ---- FUNCTION/F_GetDorPressure.TcPOU
FUNCTION F_GetDorPressure : real
VAR_INPUT
	nPressurePV:INT;
END_VAR

VAR
	Value:REAL;
END_VAR

//F_GetDorPressure := -190 * ((10 / 32767 ) * nPressurePV)+ 950;
Value:= (10.0 / 32767.0) * nPressurePV;
F_GetDorPressure := (190* (Value) ) - 190;

END_FUNCTION

// ---- POUs/P90_Interlock.TcPOU
PROGRAM P90_Interlock
VAR
	bRecipeRunning 		: BOOL;
	RecipeStopped 		: BOOL;
	ManualOperation 	: BOOL;
	bInductionHeaterMC	: BOOL;
	bThermalBathMC		: BOOL;
	bVacuumPumpMC 		: BOOL;
	bLineHeaterMC 		: BOOL; 

	bRecipeStartAvailable	: BOOL;
	bReactorOpenEnable		: BOOL;
	bHeaterOnEnable			: BOOL;
	bPumpOnEnable			: BOOL;
	
	bDorOnEnable			: BOOL;
	bDorOffEnable			: BOOL;
	bOpenEnableTemp			: BOOL;
	bOpenEnablePress		: BOOL;	
	
	bPowerResetSwitch		: BOOL;
	bMainPowerMonitor		: BOOL;

	AlarmTrig				: BOOL;
	WarningTrig				: BOOL;
	bMaintKey				: BOOL;
	bGasStateProcess		: BOOL; // True가 모든 벨브가 닫힌 상태
	bGasStateSource			: BOOL;// True가 모든 벨브가 닫힌 상태
	bGasStateVent			: BOOL;// True가 모든 벨브가 닫힌 상태

	bPowerResetLED			: BOOL;
	bUPSMode				: BOOL;
	tAlarmDelay_A			: TIME; //아날로그 디바이스 지연시간
	tAlarmDelay_D			: TIME; //디지털 디바이스 지연시간
	
	fbDeviationCheck		:ARRAY[1..29] OF FB_DeviationCheck;
	wDeviceAlarmEnable		: DWORD;
	wDeviceWarningEnable	: DWORD;
	bDeviationAlarm			: BOOL;
	bDeviationWarning		: BOOL;
	wDeviationAlarm			: DWORD;
	wDeviationWarning		: DWORD;

	wLimitAlarmEnable		: DWORD;
	wLimitWarningEnable		: DWORD;
	bLimitAlarm				: BOOL;
	bLimitWarning			: BOOL;
	wLimitAlarm				: DWORD;
	wLimitWarning			: DWORD;
	
	wAlarmEnable			: DWORD;
	wWarningEnable			: DWORD;

	bFaultAlarm				: BOOL;
	bFaultWarning			: BOOL;
	wAlarm					: DWORD;
	wWarning				: DWORD;
		
	bAlarmEnable			: BOOL;
	bWarningEnable			: BOOL;
	bDeviceCurrentAlarmState	: BOOL;
	bDeviceCurrentWarningState 	: BOOL;
	fDeviceCurrentValue			: REAL;
	fDeviceAlarmTreshold		: REAL;
	fDeviceWarningTreshold		: REAL;
	
	i	: INT;
	j 	: INT;

END_VAR

(* Read from Device*)
_DigitalInput();

bGasStateProcess := F_StateValve_Process();  // True 가  Close 상태
bGasStateSource := F_StateValve_Process_Source(); // Process gas safety / Source Carier Gas
bGasStateVent := F_State_All_Valve_Vent();//벤트 가능 조건

GVL_IO.aInterlock[1].10 := bRecipeStartAvailable;
GVL_IO.aInterlock[1].11 := bReactorOpenEnable;
GVL_IO.aInterlock[1].12 := bPumpOnEnable;
//알람 지연 시간 변환
tAlarmDelay_A := REAL_TO_TIME(GVL_IO.aInterlockSet[3]*1000); // UI Setting Analog Delay Time Value(Miliseconde)
tAlarmDelay_D := REAL_TO_TIME(GVL_IO.aInterlockSet[4]*1000); // UI Setting Analog Delay Time Value(Miliseconde)

IF bMaintKey THEN //bMaintKey 변경
	GVL_IO.nCaseSignalTower	:= 4; //Signal Tower Blue - Maintenance
	GVL_COMMAND_FROM_UI.CMD_HEATER_MAIN_MC_ON := GVL_IO.aOutputCmd[1].0;
	GVL_COMMAND_FROM_UI.CMD_THERMAL_BACH_MC_ON:=GVL_IO.aOutputCmd[1].1;
	GVL_COMMAND_FROM_UI.CMD_VACUUM_PUMP_MC_ON:=GVL_IO.aOutputCmd[1].2;
	GVL_COMMAND_FROM_UI.CMD_LINE_HEATER_MC_ON:=GVL_IO.aOutputCmd[1].3;
ELSE
	_100_Alarm_Pressure_Low();
	_101_Alarm_MFC_EPC();
	_102_Alarm_Reactor_Temp_Pre_Rotation();
	_103_Alarm_Reactor_OverPre_Temp();
	_104_Alarm_Utility();	
	_105_Alarm_Utility_Parts();
	_Button_Reset_Warning();
END_IF

_01_Enable_RunRecipe();
_02_Enable_Reactor_Open_Dor_Off();
_03_Enable_DOR_ON();
_04_Enable_Heater_ON();
_05_Enable_OpenPressure();
_06_Enable_OpenTemp();
_07_Enable_PumpTurnOn();


(* Out to Device*)
GVL_IO.aDigitalOutputIO[3].7 := bPowerResetLED;
GVL_IO.aDigitalOutputIO[2].4 := bUPSMode;

ACTION _01_Enable_RunRecipe:
 bRecipeStartAvailable := //레시피 가능한 상태이면 TRUE
 	(AlarmTrig = FALSE) AND
 	(WarningTrig = FALSE) AND
 	(bMaintKey = FALSE ) AND
	(GVL_IO.bDORState = TRUE) AND //DOR ON 상태
// 	(RCP.userState <> 10) AND //Not Recipe Run State
 	(GVL_IO_REACTOR_CABINET.DI_03_ReactorDoorDownLimitSensor = TRUE ) AND //Cover Lower Limt
 	(bGasStateProcess = TRUE ) AND //Safety Process Gas : TRUE
 	(bGasStateSource = TRUE ) AND //Safety Source Gas : TRUE
 	(bGasStateVent = TRUE ) AND  //safety Vent Vlave : true
	(GVL_IO_VALVE.DO_00_V21PumpByPass = TRUE) AND
 	GVL_IO.nE3508_nInputManAutoBytes.0 = FALSE AND //Temperature Controller Auto : false
	GVL_DEVICE_NET_IQ_PLUS.nOutputSetType = 1 AND
	GVL_IO_REACTOR_CABINET.DI_03_CylinderAutoSwitch_Closed = TRUE ; 
	 
//jhkang 임시  on
bRecipeStartAvailable:=TRUE; 


GVL_IO.UI_INTERLOCK_CHECK_RECIPE_ENABLE.0:=(AlarmTrig = FALSE); //알람 상태 아닐것
GVL_IO.UI_INTERLOCK_CHECK_RECIPE_ENABLE.1:=(WarningTrig = FALSE); // 어닝 상태 사닐것
GVL_IO.UI_INTERLOCK_CHECK_RECIPE_ENABLE.2:=(bMaintKey = FALSE); // 메인트키 
GVL_IO.UI_INTERLOCK_CHECK_RECIPE_ENABLE.3:=(GVL_IO.bDORState = TRUE ); //DOR ON
//GVL_IO.UI_INTERLOCK_CHECK_RECIPE_ENABLE.4:=RCP.userState <> 10; // Recipe Not Running
GVL_IO.UI_INTERLOCK_CHECK_RECIPE_ENABLE.4:=GVL_IO_REACTOR_CABINET.DI_03_ReactorDoorDownLimitSensor = TRUE;  //Chamber Close
GVL_IO.UI_INTERLOCK_CHECK_RECIPE_ENABLE.5:=bGasStateProcess;  // Gas Valve Close
GVL_IO.UI_INTERLOCK_CHECK_RECIPE_ENABLE.6:=bGasStateSource; // Source Valve Close
GVL_IO.UI_INTERLOCK_CHECK_RECIPE_ENABLE.7:=bGasStateVent;//Vent Valve Close
GVL_IO.UI_INTERLOCK_CHECK_RECIPE_ENABLE.8:=(GVL_IO_VALVE.DO_00_V21PumpByPass = TRUE);  // Valve 21 open
GVL_IO.UI_INTERLOCK_CHECK_RECIPE_ENABLE.9:=GVL_IO.nE3508_nInputManAutoBytes.0 = FALSE;  // Temp Auto Mode
GVL_IO.UI_INTERLOCK_CHECK_RECIPE_ENABLE.10:=GVL_DEVICE_NET_IQ_PLUS.nOutputSetType = 1;  // Temp Auto Mode
GVL_IO.UI_INTERLOCK_CHECK_RECIPE_ENABLE.11:=GVL_IO_REACTOR_CABINET.DI_03_CylinderAutoSwitch_Closed = TRUE;  // Chamber Clamp Close
END_ACTION

ACTION _02_Enable_Reactor_Open_Dor_Off:
// DOR Off Conditions
//jhkang (GVL_IO.aInterlockEnable[1].3 = FALSE ) AND //Can Open Temperature Check
//왜 UI 에서 설정되는 Can OPen Temp / Pressure 를 확인 하는지 ? 
 
bReactorOpenEnable :=
	(AlarmTrig = FALSE) AND
	bOpenEnableTemp = TRUE AND
	bOpenEnablePress= TRUE AND
	(GVL_IO.bDORState = FALSE) AND  // DOR oFF
	(RCP.userState <> 10) AND //Not Recipe Run State
	(bGasStateProcess = TRUE ) AND //Safety Process Gas : TRUE
 	(bGasStateSource = TRUE ) AND //Safety Source Gas : TRUE
 	(bGasStateVent = TRUE ) AND  //safety Vent Vlave : true
	(GVL_IO.aInterlockEnable[1].3 = TRUE ) AND //Can Open Temperature Check
	(GVL_IO.aInterlockEnable[1].4 = TRUE ); //Can Open Pressure Check

bDorOffEnable:=
	(AlarmTrig = FALSE) AND
	bOpenEnableTemp = TRUE AND
	bOpenEnablePress= TRUE AND
//	(GVL_IO.bDORState = FALSE) AND  // DOR oFF
	(RCP.userState <> 10) AND //Not Recipe Run State
	(bGasStateProcess = TRUE ) AND //Safety Process Gas : TRUE
 	(bGasStateSource = TRUE ) AND //Safety Source Gas : TRUE
 	(bGasStateVent = TRUE ) AND  //safety Vent Vlave : true
	(GVL_IO.aInterlockEnable[1].3 = TRUE ) AND //Can Open Temperature Check
	(GVL_IO.aInterlockEnable[1].4 = TRUE ); //Can Open Pressure Check


	
GVL_IO.UI_INTERLOCK_CHECK_OPEN_REACTOR.0 := (AlarmTrig = FALSE);  //알람 상태 아닐것
GVL_IO.UI_INTERLOCK_CHECK_OPEN_REACTOR.1 := bOpenEnableTemp;  // Open Temp
GVL_IO.UI_INTERLOCK_CHECK_OPEN_REACTOR.2 := bOpenEnablePress;// Open Pressure
GVL_IO.UI_INTERLOCK_CHECK_OPEN_REACTOR.3 := GVL_IO.bDORState = FALSE; // Dor False
GVL_IO.UI_INTERLOCK_CHECK_OPEN_REACTOR.4 := RCP.userState <> 10; // Recipe Not Running
GVL_IO.UI_INTERLOCK_CHECK_OPEN_REACTOR.5 := bGasStateProcess;// Gas Valve Close
GVL_IO.UI_INTERLOCK_CHECK_OPEN_REACTOR.6 := bGasStateSource;// Source Valve Close
GVL_IO.UI_INTERLOCK_CHECK_OPEN_REACTOR.7 := bGasStateVent;// Vent Valve Close
GVL_IO.UI_INTERLOCK_CHECK_OPEN_REACTOR.8 := GVL_IO.aInterlockEnable[1].3 = TRUE; // UI 에서 Temp Interlock 설정
GVL_IO.UI_INTERLOCK_CHECK_OPEN_REACTOR.9 := GVL_IO.aInterlockEnable[1].4 = TRUE;// UI 에서 Pressure Interlock 설정
END_ACTION

ACTION _03_Enable_DOR_ON:
//jhkang Dor ON 조건 다시 확인 필요
bDorOnEnable :=	(AlarmTrig = FALSE ) AND 
				GVL_IO.isCoverClosed AND 
//				GVL_IO.bDorState = FALSE AND
				(RCP.userState <> 10) AND //Not Recipe Run State 
				GVL_IO.isPumpRunning;

GVL_IO.bDorOnEnable := bDorOnEnable;
END_ACTION

ACTION _04_Enable_Heater_ON:
bHeaterOnEnable := (AlarmTrig = FALSE ) AND 
				(GVL_IO_REACTOR_CABINET.DI_03_ReactorDoorDownLimitSensor = TRUE ) AND //Cover Lower Limt;
				GVL_IO.bDorState = TRUE AND
				(RCP.userState <> 10); //Not Recipe Run State
END_ACTION

ACTION _05_Enable_OpenPressure:
IF  GVL_IO.wIqPlus_CDG1_PV > GVL_IO.aInterlockSet[10] THEN  //Can Open Reactor Pressure
	bOpenEnablePress := TRUE;
ELSE
	bOpenEnablePress := FALSE;
END_IF
END_ACTION

ACTION _06_Enable_OpenTemp:
//jhkang Can Open Temp 가 3508 온도 맞는지?
IF  P11_E3508.wE3508_PV < GVL_IO.aInterlockSet[9] THEN  // Can Open Temp
	bOpenEnableTemp := TRUE;
ELSE
	bOpenEnableTemp := FALSE;
END_IF
END_ACTION

ACTION _07_Enable_PumpTurnOn:
bPumpOnEnable :=  // Pump ON 
	(AlarmTrig = FALSE) AND
	(GVL_IO_REACTOR_CABINET.DI_03_ReactorDoorDownLimitSensor = TRUE );
END_ACTION

ACTION _100_Alarm_Pressure_Low:
//Gas Pressure Alarm N2, H2, H2S, H2Se
FOR i := 1 TO 4 DO
	wLimitAlarmEnable := SHR(GVL_IO.aInterlockEnable[4], (i-1)); 
	wLimitWarningEnable := SHR(GVL_IO.aInterlockEnable[5], (i-1));
	GVL_SEQUENCE.fbSensorLimitCheck[i](
		bAlarmEnable := wLimitAlarmEnable.0,  // Enable 
		bWarningEnable := wLimitWarningEnable.0,
		fCurrentValue := GVL_IO.aMonitoring_PV[(i+3)], // 현재 값 
		fAlarmTreshold := GVL_IO.aInterlockSet[5],
		fWarningTreshold := GVL_IO.aInterlockSet[6],
		tAlarmDelay := tAlarmDelay_D,
		bLimitAlarm => bLimitAlarm, //알람 출력
		bLimitWarning => bLimitWarning //주의(Warning) 출력
		);	
	IF bLimitAlarm THEN		
		GVL_IO.aInterlock[1].0 := TRUE; //Alarm Trig
		GVL_IO.nCaseSignalTower := 1; // Signal Tower RED - Alarm
		//팝업 표시
		wLimitAlarm := ROR(GVL_IO.aInterlock[2], (i-1));
		wLimitAlarm.0 := TRUE;
		GVL_IO.aInterlock[2] := ROL(wLimitAlarm, (i-1));
		//대시보드 표시
		wLimitAlarm := ROR(GVL_IO.aInterlock[1], (i*2));
		wLimitAlarm.0 := TRUE;
		GVL_IO.aInterlock[1] := ROL(wLimitAlarm, (i*2));
	ELSE
		//팝업 표시
		wLimitAlarm := ROR(GVL_IO.aInterlock[2], (i-1));
		wLimitAlarm.0 := FALSE;
		GVL_IO.aInterlock[2] := ROL(wLimitAlarm, (i-1));
		//대시보드 표시
		wLimitAlarm := ROR(GVL_IO.aInterlock[1], (i*2));
		wLimitAlarm.0 := FALSE;
		GVL_IO.aInterlock[1] := ROL(wLimitAlarm, (i*2));
	END_IF
	
	IF bLimitWarning THEN		
		GVL_IO.aInterlock[1].1 := TRUE; //Warning Trig
		GVL_IO.nCaseSignalTower := 2; // Signal Tower YELLOW - Warning
		//팝업 표시
		wLimitWarning := ROR(GVL_IO.aInterlock[4], (i-1));
		wLimitWarning.0 := TRUE;
		GVL_IO.aInterlock[4] := ROL(wLimitWarning, (i-1));
		//대시보드 표시
		wLimitWarning := ROR(GVL_IO.aInterlock[1], (i*2)+1);
		wLimitWarning.0 := TRUE;
		GVL_IO.aInterlock[1] := ROL(wLimitWarning, (i*2)+1);
	ELSE
		//팝업 표시
		wLimitWarning := ROR(GVL_IO.aInterlock[4], (i-1));
		wLimitWarning.0 := FALSE;
		GVL_IO.aInterlock[4] := ROL(wLimitWarning, (i-1));
		//대시보드 표시
		wLimitWarning := ROR(GVL_IO.aInterlock[1], (i*2)+1);
		wLimitWarning.0 := FALSE;
		GVL_IO.aInterlock[1] := ROL(wLimitWarning, (i*2)+1);
	END_IF
END_FOR
END_ACTION

ACTION _101_Alarm_MFC_EPC:
//jhkang MFC ,EPC
FOR i := 1 TO 16 DO
		wDeviceAlarmEnable := SHR(GVL_IO.aInterlockEnable[2], (i+2)); //오늘쪽 쉬프트 연산
		wDeviceWarningEnable := SHR(GVL_IO.aInterlockEnable[3], (i+2));
		
		GVL_SEQUENCE.fbDeviationCheck[i](
			bAlarmEnable := wDeviceAlarmEnable.0,
			bWarningEnable := wDeviceWarningEnable.0,
			fCurrentValue := GVL_IO.aController_PV[i],
			fControlValue := LREAL_TO_REAL(GVL_IO.aController[i].rControlValue),
			fMaxValue := GVL_CONSTANT.AnalogControllerOutputVoltage,
			fAlarmTreshold := GVL_IO.aInterlockSet[1],
			fWarningTreshold := GVL_IO.aInterlockSet[2],
			tAlarmDelay := tAlarmDelay_A,
			bDeviationAlarm => bDeviationAlarm, //알람 출력
			bDeviationWarning => bDeviationWarning // 주의(Warning) 출력
			);
			
		IF bDeviationAlarm THEN
			GVL_IO.aInterlock[1].0 := TRUE; //Alarm Trig
			GVL_IO.nCaseSignalTower := 1; // Signal Tower RED - Alarm
			wDeviationAlarm := ROR(GVL_IO.aInterlock[3], (i+2));
			wDeviationAlarm.0 := TRUE;
			GVL_IO.aInterlock[3] := ROL(wDeviationAlarm, (i+2));
		ELSE
			wDeviationAlarm := ROR(GVL_IO.aInterlock[3], (i+2));
			wDeviationAlarm.0 := FALSE;
			GVL_IO.aInterlock[3] := ROL(wDeviationAlarm, (i+2));	
		END_IF
		
		IF bDeviationWarning THEN
			GVL_IO.aInterlock[1].1 := TRUE; // Warning Trig
			GVL_IO.nCaseSignalTower := 2; // Signal Tower Yellow - Warning
			wDeviationWarning := ROR(GVL_IO.aInterlock[5], (i+2));
			wDeviationWarning.0 := TRUE;
			GVL_IO.aInterlock[5] := ROL(wDeviationWarning, (i+2));
		ELSE
			wDeviationWarning := ROR(GVL_IO.aInterlock[5], (i+2));
			wDeviationWarning.0 := FALSE;
			GVL_IO.aInterlock[5] := ROL(wDeviationWarning, (i+2));
		END_IF
	END_FOR
END_ACTION

ACTION _102_Alarm_Reactor_Temp_Pre_Rotation:
//jhkang Reactor Temp , Pressure ,Rotation

FOR i := 1 TO 3 DO
		wDeviceAlarmEnable := SHR(GVL_IO.aInterlockEnable[2], (i-1)); //오늘쪽 쉬프트 연산
		wDeviceWarningEnable := SHR(GVL_IO.aInterlockEnable[3], (i-1));
		
		GVL_SEQUENCE.fbDeviationCheck_Reactor[i](
			bAlarmEnable := wDeviceAlarmEnable.0,
			bWarningEnable := wDeviceWarningEnable.0,
			fCurrentValue := GVL_IO.aController_PV[i+16],
			fControlValue := LREAL_TO_REAL(GVL_IO.aController[i+16].rControlValue),
			fMaxValue := GVL_IO.aReactorMaxValue[i],
			fAlarmTreshold := GVL_IO.aInterlockSet[1],
			fWarningTreshold := GVL_IO.aInterlockSet[2],
			tAlarmDelay := tAlarmDelay_A,
			bDeviationAlarm => bDeviationAlarm, //알람 출력
			bDeviationWarning => bDeviationWarning // 주의(Warning) 출력
			);
			
		IF bDeviationAlarm THEN
			GVL_IO.aInterlock[1].0 := TRUE; //Alarm Trig
			GVL_IO.nCaseSignalTower := 1; // Signal Tower RED - Alarm
			wDeviationAlarm := ROR(GVL_IO.aInterlock[3], (i-1));
			wDeviationAlarm.0 := TRUE;
			GVL_IO.aInterlock[3] := ROL(wDeviationAlarm, (i-1));
		ELSE
			wDeviationAlarm := ROR(GVL_IO.aInterlock[3], (i-1));
			wDeviationAlarm.0 := FALSE;
			GVL_IO.aInterlock[3] := ROL(wDeviationAlarm, (i-1));	
		END_IF
		
		IF bDeviationWarning THEN
			GVL_IO.aInterlock[1].1 := TRUE; // Warning Trig
			GVL_IO.nCaseSignalTower := 2; // Signal Tower Yellow - Warning
			wDeviationWarning := ROR(GVL_IO.aInterlock[5], (i-1));
			wDeviationWarning.0 := TRUE;
			GVL_IO.aInterlock[5] := ROL(wDeviationWarning, (i-1));
		ELSE
			wDeviationWarning := ROR(GVL_IO.aInterlock[5], (i-1));
			wDeviationWarning.0 := FALSE;
			GVL_IO.aInterlock[5] := ROL(wDeviationWarning, (i-1));
		END_IF
	END_FOR
END_ACTION

ACTION _103_Alarm_Reactor_OverPre_Temp:

//Over Temp Over Pressure
FOR i := 1 TO 2 DO
	CASE i OF
		
		1: //Susceptor Over Temperature
			bAlarmEnable := GVL_IO.aInterlockEnable[4].4;
			bWarningEnable := GVL_IO.aInterlockEnable[5].4;
			fDeviceCurrentValue := P11_E3508.wE3508_PV;
			fDeviceAlarmTreshold := GVL_IO.aInterlockSet[7];
			fDeviceWarningTreshold := (GVL_IO.aInterlockSet[7] * 0.9); // 90% 이상 warning 
		
		2: //Reactor Over Pressure Alarm
			bAlarmEnable := GVL_IO.aInterlockEnable[4].5;
			bWarningEnable := GVL_IO.aInterlockEnable[5].5;
			fDeviceCurrentValue := GVL_IO.wIqPlus_CDG1_PV;
			fDeviceAlarmTreshold := GVL_IO.aInterlockSet[8];
			fDeviceWarningTreshold := (GVL_IO.aInterlockSet[8] * 0.9); //
			
	END_CASE
	
	GVL_SEQUENCE.fbSensorOverLimitCheck[i](
		bAlarmEnable	 := bAlarmEnable,  // Enable 
		bWarningEnable	 := bWarningEnable,
		fCurrentValue  := fDeviceCurrentValue, // 현재 값 
		fAlarmTreshold	 := fDeviceAlarmTreshold,
		fWarningTreshold  := fDeviceWarningTreshold,
		tAlarmDelay := tAlarmDelay_D,
		bAlarm => bLimitAlarm, //알람 출력
		bWarning => bLimitWarning //주의(Warning) 출력
		);
	
		IF bLimitAlarm THEN
			GVL_IO.aInterlock[1].0 := TRUE; //Alarm Trig
			GVL_IO.nCaseSignalTower := 1; // Signal Tower RED - Alarm
			wDeviationAlarm := ROR(GVL_IO.aInterlock[2], (i+3));
			wDeviationAlarm.0 := TRUE;
			GVL_IO.aInterlock[2] := ROL(wDeviationAlarm, (i+3));
		ELSE
			wDeviationAlarm := ROR(GVL_IO.aInterlock[2], (i+3));
			wDeviationAlarm.0 := FALSE;
			GVL_IO.aInterlock[2] := ROL(wDeviationAlarm, (i+3));	
		END_IF
		
		IF bLimitWarning THEN
			GVL_IO.aInterlock[1].1 := TRUE; // Warning Trig
			GVL_IO.nCaseSignalTower := 2; // Signal Tower Yellow - Warning
			wDeviationWarning := ROR(GVL_IO.aInterlock[4], (i+3));
			wDeviationWarning.0 := TRUE;
			GVL_IO.aInterlock[4] := ROL(wDeviationWarning, (i+3));
		ELSE
			wDeviationWarning := ROR(GVL_IO.aInterlock[4], (i+3));
			wDeviationWarning.0 := FALSE;
			GVL_IO.aInterlock[4] := ROL(wDeviationWarning, (i+3));
		END_IF
END_FOR
END_ACTION

ACTION _104_Alarm_Utility:
	//Device Fault Check - Pneumatic, Heater, Pump, Motor, GC Door, RC Door
	FOR i := 1 TO 7 DO
		CASE i OF
			1: //CDA Alarm Switch (Pneumatic)
				bAlarmEnable := GVL_IO.aInterlockEnable[4].6;
				bWarningEnable := GVL_IO.aInterlockEnable[5].6;
				bDeviceCurrentAlarmState := NOT GVL_IO.aInputState[1].3;
				bDeviceCurrentWarningState := NOT GVL_IO.aInputState[1].3;
				
			2: //Cooling Water Switch
				bAlarmEnable := GVL_IO.aInterlockEnable[4].7;
				bWarningEnable := GVL_IO.aInterlockEnable[5].7;
				bDeviceCurrentAlarmState := NOT GVL_IO.aInputState[1].4;
				bDeviceCurrentWarningState := NOT GVL_IO.aInputState[1].4;
				
			3: //Rotatin Motor Fault
				bAlarmEnable := GVL_IO.aInterlockEnable[4].8;
				bWarningEnable := GVL_IO.aInterlockEnable[5].8;
				bDeviceCurrentAlarmState :=  GVL_IO.aInputState[1].7;
				bDeviceCurrentWarningState :=  GVL_IO.aInputState[1].7;
				
			4: //Vacuum Pump Fault
				bAlarmEnable := GVL_IO.aInterlockEnable[4].9;
				bWarningEnable := GVL_IO.aInterlockEnable[5].9;
				bDeviceCurrentAlarmState := NOT GVL_IO.aInputState[1].10;
				bDeviceCurrentWarningState := NOT GVL_IO.aInputState[1].9;
				
			5: //Gas Cabinet Door Open
				bAlarmEnable := GVL_IO.aInterlockEnable[4].10;
				bWarningEnable := GVL_IO.aInterlockEnable[5].10;
				bDeviceCurrentAlarmState := NOT GVL_IO.aInputState[1].15;
				bDeviceCurrentWarningState := NOT GVL_IO.aInputState[1].15;
			6: //Reactor Cabinet Door Open
				bAlarmEnable := GVL_IO.aInterlockEnable[4].11;
				bWarningEnable := GVL_IO.aInterlockEnable[5].11;
				bDeviceCurrentAlarmState := NOT GVL_IO.aInputState[1].13;
				bDeviceCurrentWarningState := NOT GVL_IO.aInputState[1].13;
				
			7: //DOR Fault
				bAlarmEnable := GVL_IO.aInterlockEnable[4].12;
				bWarningEnable := GVL_IO.aInterlockEnable[5].12;
				
				IF (GVL_IO.nDorOperationError = 1) THEN
					bDeviceCurrentAlarmState := TRUE;
				ELSE
					bDeviceCurrentAlarmState := FALSE;
				END_IF
				IF (GVL_IO.nDorOperationError = 2) OR (GVL_IO.nDorOperationError = 3) THEN
					bDeviceCurrentWarningState := TRUE;
					bDeviceCurrentAlarmState:=TRUE;
				ELSE
					bDeviceCurrentWarningState := FALSE;
					bDeviceCurrentAlarmState:=FALSE;
				END_IF
		END_CASE

		GVL_SEQUENCE.fbFaultCheck[i](
			bAlarmEnable := bAlarmEnable,
			bWarningEnable := bWarningEnable,
			bCurrentAlarmState := bDeviceCurrentAlarmState,
			bCurrentWarningState := bDeviceCurrentWarningState,
			tAlarmDelay := tAlarmDelay_D,
			bAlarm => bFaultAlarm,
			bWarning => bFaultWarning
			);
			
		IF bFaultAlarm THEN
			GVL_IO.aInterlock[1].0 := TRUE; //Alarm Trig
			GVL_IO.nCaseSignalTower := 1; // Signal Tower RED - Alarm
			//팝업 표시
			wAlarm := ROR(GVL_IO.aInterlock[2], (i+5));
			wAlarm.0 := TRUE;
			GVL_IO.aInterlock[2] := ROL(wAlarm, (i+5));
		END_IF
		IF bFaultWarning THEN
			GVL_IO.aInterlock[1].1 := TRUE; //Warning Trig
			GVL_IO.nCaseSignalTower := 2; // Signal Tower YELLOW - Warning
			//팝업 표시
			wAlarm := ROR(GVL_IO.aInterlock[4], (i+5));
			wAlarm.0 := TRUE;
			GVL_IO.aInterlock[4] := ROL(wAlarm, (i+5));
		END_IF
	END_FOR
END_ACTION

ACTION _105_Alarm_Utility_Parts:
//SMPS,Circuit Power , Gas Detector ,
	FOR i := 1 TO 4 DO
		CASE i OF
			1: //SMPS
				bAlarmEnable := GVL_IO.aInterlockEnable[4].13;
				bDeviceCurrentAlarmState := GVL_IO.aInputState[2].5 OR 
											GVL_IO.aInputState[2].6 OR 
											GVL_IO.aInputState[2].7 OR 
											GVL_IO.aInputState[2].8;
			2: //Circuit Power
				bAlarmEnable := GVL_IO.aInterlockEnable[4].14;
				bDeviceCurrentAlarmState := GVL_IO.aInputState[2].13 = FALSE  OR  
											GVL_IO.aInputState[2].14 = FALSE  OR
											GVL_IO.aInputState[2].15 = FALSE  OR
											GVL_IO.aInputState[3].0 = FALSE  OR 
											GVL_IO.aInputState[3].1 = FALSE  OR
											GVL_IO.aInputState[3].2  = FALSE;
				//bDeviceCurrentAlarmState 가 true 면 알람 상태 
				
		//GVL_IO.aInputState[2].13:= GVL_IO_GAS_CABINET.DI_02_RotationMotorCP;
		//GVL_IO.aInputState[2].14:= GVL_IO_GAS_CABINET.DI_02_CoverLiftMotorCP;
		//GVL_IO.aInputState[2].15:= GVL_IO_GAS_CABINET.DI_02_T_VCP;
		
		//GVL_IO.aInputState[3].0:= GVL_IO_GAS_CABINET.DI_03_GasDetectorCP;
		//GVL_IO.aInputState[3].1:= GVL_IO_GAS_CABINET.DI_03_CabinetLampsCP;
		//GVL_IO.aInputState[3].2:= GVL_IO_GAS_CABINET.DI_03_MFCPowerCP;

			3: //Gas Detector
				bAlarmEnable := GVL_IO.aInterlockEnable[4].15;
				bDeviceCurrentAlarmState := GVL_IO.aInputState[3].11 AND GVL_IO.aInputState[3].12 AND GVL_IO.aInputState[3].13 AND GVL_IO.aInputState[3].14;
				

		//GVL_IO.aInputState[3].11:= GVL_IO_GAS_CABINET.DI_04_GasDetectorH2;
		//GVL_IO.aInputState[3].12:= GVL_IO_GAS_CABINET.DI_04_GasDetectorH2S;
		//GVL_IO.aInputState[3].13:= GVL_IO_GAS_CABINET.DI_04_GasDetectorH2Se;
		//GVL_IO.aInputState[3].14:= GVL_IO_GAS_CABINET.DI_04_FireSensor;
			4: // External Alarm
				bAlarmEnable := GVL_IO.aInterlockEnable[4].16;
				bDeviceCurrentAlarmState := GVL_IO.aInputState[3].14 AND GVL_IO.aInputState[3].15 AND GVL_IO.aInputState[4].0 AND GVL_IO.aInputState[4].1 AND GVL_IO.aInputState[4].2
														AND GVL_IO.aInputState[4].3 AND GVL_IO.aInputState[4].4;
				
						
		//GVL_IO.aInputState[3].14:= GVL_IO_GAS_CABINET.DI_04_FireSensor;
		//GVL_IO.aInputState[3].15 := GVL_IO_GAS_CABINET.DI_04_ExternalScrubberFault;
		//GVL_IO.aInputState[4].0 := GVL_IO_GAS_CABINET.DI_05_ExternalH2GasCabinetFault;
		//GVL_IO.aInputState[4].1 := GVL_IO_GAS_CABINET.DI_05_ExternalH2SGasCabinetFault;
		//GVL_IO.aInputState[4].2 := GVL_IO_GAS_CABINET.DI_05_ExternalH2SeGasCabinetFault;
		//GVL_IO.aInputState[4].3 := GVL_IO_GAS_CABINET.DI_05_ExternalUserInputAlarm;

		END_CASE

		GVL_SEQUENCE.fbFaultCheck_Utility_CP[i](
			bAlarmEnable := bAlarmEnable,
			bWarningEnable := FALSE,
			bCurrentAlarmState := bDeviceCurrentAlarmState,
			bCurrentWarningState := FALSE,
			tAlarmDelay := tAlarmDelay_D,
			bAlarm => bFaultAlarm,
			bWarning => bFaultWarning
			);
			
		IF bFaultAlarm THEN
			GVL_IO.aInterlock[1].0 := TRUE; //Alarm Trig
			GVL_IO.nCaseSignalTower := 1; // Signal Tower RED - Alarm
			//팝업 표시
			wAlarm := ROR(GVL_IO.aInterlock[2], (i+13));
			wAlarm.0 := TRUE;
			GVL_IO.aInterlock[2] := ROL(wAlarm, (i+13));
		END_IF
	END_FOR
END_ACTION

ACTION _Button_Reset_Warning:
IF GVL_IO.aInterlockEnable[1].0 THEN //알람 리셋 버턴을 눌렀을 때
	GVL_IO.aInterlock[1].0 := FALSE; //Alarm Trig Reset
	GVL_IO.aInterlockEnable[1].0 := FALSE; //버턴 초기화
	GVL_IO.nCaseSignalTower := 4; // Signal Tower Blue - Idle
END_IF
IF GVL_IO.aInterlockEnable[1].1 THEN //주의 리셋 버턴을 눌렀을 때
	GVL_IO.aInterlock[1].1 := FALSE; //Warmomg Trig Reset
	GVL_IO.aInterlockEnable[1].1 := FALSE; //버턴 초기화
	GVL_IO.nCaseSignalTower := 4; // Signal Tower Blue - Idle
END_IF
END_ACTION

ACTION _DigitalInput:
bMaintKey := GVL_IO_REACTOR_CABINET.DI_01_MaintenanceModeKey;
bPowerResetSwitch := GVL_IO_GAS_CABINET.DI_01_ResetButton;
//jhkang Main Power Monitor 가 뭔가 ? 
//7. 순간정전 되었다가 전기가 다시 살아 났을 때,
// UPS는 전원이 살아있고, 히터, 펌프, bath는 전기가 나갔을 때 (아직 명확한 로직이 없음)
bMainPowerMonitor := GVL_IO.aDigitalInputIO[7].5; /// ??????? 이게 뭐지 ?
END_ACTION

END_PROGRAM

// ---- POUs/FB_DeviationCheck.TcPOU
//*********************************************************************
// Function Block: FB_DeviationCheck
// Description: 각 디바이스의 편차 초과 알람을 처리합니다.
// bEnable이 TRUE일 때만 알람 로직이 활성화됩니다.
//*********************************************************************
FUNCTION_BLOCK FB_DeviationCheck
VAR_INPUT
	bAlarmEnable	: BOOL; // 디바이스 활성화/비활성화 (TRUE = 활성화)
	bWarningEnable	: BOOL;
	fCurrentValue 	: REAL; //현재값
	fControlValue 	: REAL; //제어값
	fMaxValue		: REAL; //최대값
	fAlarmTreshold	: REAL; // 알람 편차 허용 임계값
	fWarningTreshold : REAL; // 경고 편차 허용 임계값
	tAlarmDelay		: TIME; //알람 지연 시간
END_VAR
VAR_OUTPUT
	bDeviationAlarm		: BOOL; //편차 알람 발생
	bDeviationWarning 	: BOOL; //편차 경고 발생
	fDeviationAlarm		: REAL; // 현재 편차(참고용)
	fDeviationWarning	: REAL; 
END_VAR
VAR
	// 내부 변수 (인스턴스별로 독립적)
	fbDeviationAlarmTimer 		: TON;
	fbDeviationWarningTimer 	: TON; 
	bDeviationAlarmCondition 	: BOOL;
	bDeviationWarningCondition 	: BOOL; 
END_VAR

// bAlarmEnable이 TRUE일 때만 알람 로직 실행
IF bAlarmEnable AND (fMaxValue <> 0) THEN
	fDeviationAlarm :=ABS(fCurrentValue - fControlValue)/fMaxValue * 100; //편차 계산(%)
	//편차 알람 로직(지연 시간 적용)
	IF fDeviationAlarm > fAlarmTreshold THEN
		bDeviationAlarmCondition := TRUE;
	ELSE
		bDeviationAlarmCondition := FALSE;
	END_IF
	fbDeviationAlarmTimer(IN:=bDeviationAlarmCondition, PT:=tAlarmDelay);
	bDeviationAlarm := fbDeviationAlarmTimer.Q;
ELSE
	// bEnable이 FALSE일 경우, 모든 알람 및 타이머를 비활성화/리셋
    // Q 출력을 FALSE로 강제하고, IN 입력을 FALSE로 설정하여 타이머를 리셋합니다.
	bDeviationAlarm := FALSE;
	fbDeviationAlarmTimer(IN := FALSE, PT := tAlarmDelay); // 타이머 리셋
	bDeviationAlarmCondition := FALSE; // 조건 플래그도 리셋
	fDeviationAlarm := 0.0; // 편차 값도 0으로 초기화 (선택 사항)
END_IF

// bWarningEnable이 TRUE일 때만 알람 로직 실행
IF bWarningEnable AND (fMaxValue <> 0) THEN
	//편차 계산(%)
	fDeviationWarning :=ABS(fCurrentValue - fControlValue)/fMaxValue * 100;
	//편차 알람 로직(지연 시간 적용)
	IF (fDeviationWarning > fWarningTreshold) AND (fDeviationWarning <= fAlarmTreshold) THEN
		bDeviationWarningCondition := TRUE;
	ELSE
		bDeviationWarningCondition := FALSE;
	END_IF
	fbDeviationWarningTimer(IN:=bDeviationWarningCondition, PT:=tAlarmDelay);
	bDeviationWarning := fbDeviationWarningTimer.Q;
ELSE
	// bEnable이 FALSE일 경우, 모든 알람 및 타이머를 비활성화/리셋
    // Q 출력을 FALSE로 강제하고, IN 입력을 FALSE로 설정하여 타이머를 리셋합니다.
	bDeviationWarning := FALSE;
	fbDeviationWarningTimer(IN := FALSE, PT := tAlarmDelay); // 타이머 리셋
	bDeviationWarningCondition := FALSE; // 조건 플래그도 리셋
	fDeviationWarning := 0.0; // 편차 값도 0으로 초기화 (선택 사항)
END_IF

END_FUNCTION_BLOCK

// ---- POUs/P11_E3508.TcPOU
PROGRAM P11_E3508
VAR
	wControlValue			: WORD;
	wPowerRateSetValue		: WORD;	
	bOutputManAuto 			: BOOL; // Command 0:Auto, 1:Manual Mode
	
	bHeaterOn				: BOOL := FALSE; //to PSTEK
	bHeaterReset			: BOOL; //to PSTEK

	bAlarmState_E3508 		: BOOL; //Alarm or Sensor Break Signal
	bManAuto_E3508 			: BOOL; //State, 0:Manual, 1:Auto

	isHeaterReady			: BOOL; //Close : Ready
	isHeaterRun				: BOOL; //Close : Running, Open : Stop
	isHeaterFault			: BOOL; //Close : Falut, Open : Normal
	//isInductionHeaterErr	: BOOL; //Power Supply
	bInductionHeaterCB		: BOOL;
	//Input from E3508 Controller
//	aInputPVBytes AT %I* 		: ARRAY[1..2]OF USINT; //Input Process Values
//	aInputSVBytes AT %I* 		: ARRAY[1..2]OF USINT; //Input Set Values
//	aInputTVBytes AT %I* 		: ARRAY[1..2]OF USINT; //Input Target Valuse
//	aInputCVBytes AT %I* 		: ARRAY[1..2]OF USINT; //Induction Heter Controlled Values
//	aInputProportional AT %I* 	: ARRAY[1..2]OF USINT; //PID - Proportional Band
//	aInputIntegral AT %I* 		: ARRAY[1..2]OF USINT; //PID - Integral Time
//	aInputDerivative AT %I* 	: ARRAY[1..2]OF USINT; //PID - Derivative Time 
//	nInputAlarmBytes AT %I* 	: USINT; // Alarm State
//	nInputManAutoBytes AT %I* 	: USINT; // ManAuto State
	
	wE3508_PV				: WORD;
	wE3508_SV				: WORD;
	wE3508_PowerRate		: WORD; //To Induction Heater Control Values
	wE3508_P				: WORD; //PID Parameter P
	wE3508_I				: WORD; //PID Parameter I
	wE3508_D				: WORD; //PID Parameter D
	//Output to E3508 Controller
	wOutputSVBytes 				: outWord;
	wOutputPowerSVBytes 		: outWord;

END_VAR

//Induction Heater & Temperature Controller & Thermo Couple(R-Type)
//Maker: PSTEK, Eurotherm
//Model: 3508
//Temperature Range: 0 ~ 12000℃

(* Command *)
bHeaterOn := GVL_COMMAND_FROM_UI.CMD_HEATER_MAIN_MC_ON;


GVL_DEVICE_NET_E3508.nOutputManAutoBytes[1].0 := GVL_COMMAND_FROM_UI.CMD_E3508_MAN_AUTO; //Temp Controller Mode Command(*True:manual   False:auto*)

(* Read from Power Distribution Pannel *)
bInductionHeaterCB		:= GVL_IO_GAS_CABINET.DI_02_GraphiteHeaterELCB;

(* Read from E3508 Device Value *)
wE3508_PV				:= USINT_TO_WORD_Bit(GVL_DEVICE_NET_E3508.aInputPVBytes[1], GVL_DEVICE_NET_E3508.aInputPVBytes[2]);
wE3508_SV				:= USINT_TO_WORD_Bit(GVL_DEVICE_NET_E3508.aInputSVBytes[1], GVL_DEVICE_NET_E3508.aInputSVBytes[2]);
wE3508_PowerRate		:= USINT_TO_WORD_Bit(GVL_DEVICE_NET_E3508.aInputActiveOut[1], GVL_DEVICE_NET_E3508.aInputActiveOut[2]); //divided to 10

wE3508_P 				:= USINT_TO_WORD_Bit(GVL_DEVICE_NET_E3508.aInputProportional[1], GVL_DEVICE_NET_E3508.aInputProportional[2]);
wE3508_I 				:= USINT_TO_WORD_Bit(GVL_DEVICE_NET_E3508.aInputIntegral[1], GVL_DEVICE_NET_E3508.aInputIntegral[2]);
wE3508_D 				:= USINT_TO_WORD_Bit(GVL_DEVICE_NET_E3508.aInputDerivative[1], GVL_DEVICE_NET_E3508.aInputDerivative[2]);

//Temp Controller Alarm
GVL_IO.aInputState[5].9:= GVL_DEVICE_NET_E3508.aInputAlarmStatus[1] > 0 OR GVL_DEVICE_NET_E3508.aInputAlarmStatus[2] > 0 ;

//bAlarmState_E3508 		:= nInputAlarmBytes.7;

//GVL_IO.aMonitoring_PV[11] := WORD_TO_REAL(wE3508_PowerRate)*0.1; //divided to 10 PowerRate

(* Read from Induction Heater Value *)

// Interface with other PRGs
wControlValue			:= GVL_IO.wE3508_CV;
GVL_IO.wE3508_PV		:= wE3508_PV;

(* Write to E3508 Device Value *)
// Operation Mode
// bOutputManAuto := GVL_IO.aOutputCmd[1].11; //Temp Controller Mode Command
// nOutputManAutoBytes.0 	:= GVL_IO.aOutputCmd[1].11; //Command

IF GVL_DEVICE_NET_E3508.aInputManAutoBytes[1].0 THEN // Read form E3508 Mode, 0:Man 1:Auto
	wOutputPowerSVBytes 	:= WORD_TO_USINT_Bit(wControlValue*10); //multiple to 10, Power Reate Set Value
	GVL_DEVICE_NET_E3508.aOutputPowerBytes[1] 	:= wOutputPowerSVBytes.Lower;
	GVL_DEVICE_NET_E3508.aOutputPowerBytes[2] 	:= wOutputPowerSVBytes.Upper;
ELSE
	wOutputSVBytes 			:= WORD_TO_USINT_Bit(wControlValue); // Temperature Set Value
	GVL_DEVICE_NET_E3508.aOutputSVBytes[1] 		:= wOutputSVBytes.Lower;
	GVL_DEVICE_NET_E3508.aOutputSVBytes[2] 		:= wOutputSVBytes.Upper;
END_IF

(* Write to Induction Heater Value *)
GVL_IO_GAS_CABINET.DO_07_GraphiteHeaterMC := bHeaterOn;
//GVL_IO.aDigitalOutputIO[2].1 := bHeaterReset;
GVL_IO.nE3508_nInputManAutoBytes := GVL_DEVICE_NET_E3508.aInputManAutoBytes[1]; //State


GVL_DEVICE_NET_E3508.aOutputThreshold[1]:=232;
GVL_DEVICE_NET_E3508.aOutputThreshold[2]:=3;

END_PROGRAM

// ---- POUs/P12_IQ_PLUS.TcPOU
PROGRAM P12_IQ_PLUS
VAR
	wControlValue 		: WORD := 760;//Pressure Set Value
	wCDG1_PV 			: WORD; //CD2 Current Pressure
	wCDG2_PV 			: WORD; //CD2 Current Pressure
	bVacuumPumpCB		: BOOL;
	bThrottleValveCP	: BOOL;

	//nInputStatus
	ingPressureControl 		: BOOL;
	ingPositionControl 		: BOOL;
	isValveOpen 			: BOOL;
	isValveNotInitialized 	: BOOL;	
	isValveClosed 			: BOOL;
	isValveFaultState 		: BOOL;
	ingValveInitializing 	: BOOL;
	ingHoldState 			: BOOL;
	isPressureControl:BOOL;
	
	// Vacuum Pump Status
	isPumpFault				: BOOL;
	isPumpWarning			: BOOL;
	isPumpAlarm				: BOOL;
	isFBRunning				: BOOL;
 	isPumpRunning			: BOOL;
	//wSetPoint 			: WORD; //Set Point
	nTValveMode 		: USINT := 0; //Valve Mode
	bPumpOn				: BOOL;
	bPumpReset			: BOOL;	//Input from IQ-PLUS Throttle Valve
	
	wTypedControlValue 	: WORD;
	wOutputSVBytes : outWord; //Word to Byte variable
	nSetType 			: USINT; //1:Pressure Conrol, 2:Position Control
	
	wByteCDG1_PV 			: WORD; //CDG1 Current Pressure, Not Used
	wByteCDG2_PV 			: WORD; //CDG2 Current Pressure
	wByteValvePosition_PV : WORD; //Current Valve Position (0~100%)
	nInputStatusOld : USINT := 9; //Value Change Monitoring, First Temp value
	wByteValvePosition_PV_Monitoring: WORD;
	CDG1_RealValue: REAL;
	nOutputSetType:USINT; //1:Pressure Conrol, 2:Position Control
	CDG_1_Value_RealType: REAL;
END_VAR

VAR CONSTANT
	//Conversion Parameter
	SetPointFactor : REAL := 327.67; //Range 0~7FFFh
	PressureFactor : REAL := 24.576;	//Range 0~6000h
END_VAR

//Model : IQ Plus 
//Pressure Range : 0 ~ 1,000 Torr
IF GVL_COMMAND_FROM_UI.CMD_THROTTLE_PRESSURE_POSITION_MODE THEN //true: Pressure False:Position
	GVL_DEVICE_NET_IQ_PLUS.nOutputSetType := 1; // Pressure Control
ELSE
	GVL_DEVICE_NET_IQ_PLUS.nOutputSetType := 2; // Position Control
END_IF

nSetType := GVL_DEVICE_NET_IQ_PLUS.nOutputSetType;
nOutputSetType:=nSetType;


_DIgitalInput();
_CalData();
_DigitalOutput();


nTValveMode := WORD_TO_USINT(GVL_IO.aOutputCmd[2]); //Throttle Valve Mode Setting 0:Normal 1:Close 2:Open 3:Hold 4:Reset

